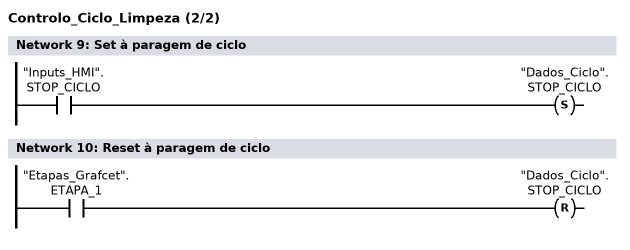
   RUNG wire#powerrail
      Contact( "Inputs_HMI".STOP_CICLO )
      S_Coil( "Dados_Ciclo".STOP_CICLO )
   END_RUNG
   // the same network as SCL:
   IF "Inputs_HMI".STOP_CICLO THEN "Dados_Ciclo".STOP_CICLO := TRUE; END_IF;
END_REGION

REGION Network 10: Reset à paragem de ciclo
   RUNG wire#powerrail
      Contact( "Etapas_Grafcet".ETAPA_1 )
      R_Coil( "Dados_Ciclo".STOP_CICLO )
   END_RUNG
   // the same network as SCL:
   IF "Etapas_Grafcet".ETAPA_1 THEN "Dados_Ciclo".STOP_CICLO := FALSE; END_IF;
END_REGION
END_FUNCTION

FUNCTION "Controlo_Pressostatos" : Void   // FC8, LAD
TITLE = Ao fim de 30s indica que atingiu setpoint de pressão
{ S7_Optimized_Access := 'TRUE' }
VERSION : 0.1
// stored: AutoNumber true, IsIECCheckEnabled false, SetENOAutomatically false, UDAEnableTagReadback false
BEGIN

REGION Network 1: Pressostato Filtro 1
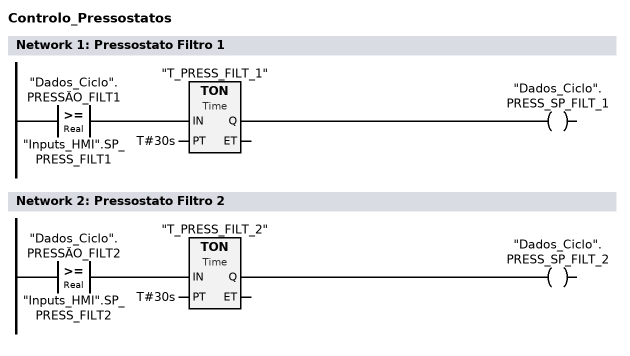
   RUNG wire#powerrail
      { S7_Templates := "SrcType := Real" } GE_Contact(in1 := "Dados_Ciclo".PRESSÃO_FILT1, in2 := "Inputs_HMI".SP_PRESS_FILT1)
      { S7_Templates := "time_type := Time" } "T_PRESS_FILT_1".TON(pt := T#30s, et =>)
      Coil( "Dados_Ciclo".PRESS_SP_FILT_1 )
   END_RUNG
   // the same network as SCL:
   "T_PRESS_FILT_1".TON(IN := "Dados_Ciclo".PRESSÃO_FILT1 >= "Inputs_HMI".SP_PRESS_FILT1, PT := T#30s);
   "Dados_Ciclo".PRESS_SP_FILT_1 := "T_PRESS_FILT_1".Q;
END_REGION

REGION Network 2: Pressostato Filtro 2
   RUNG wire#powerrail
      { S7_Templates := "SrcType := Real" } GE_Contact(in1 := "Dados_Ciclo".PRESSÃO_FILT2, in2 := "Inputs_HMI".SP_PRESS_FILT2)
      { S7_Templates := "time_type := Time" } "T_PRESS_FILT_2".TON(pt := T#30s, et =>)
      Coil( "Dados_Ciclo".PRESS_SP_FILT_2 )
   END_RUNG
   // the same network as SCL:
   "T_PRESS_FILT_2".TON(IN := "Dados_Ciclo".PRESSÃO_FILT2 >= "Inputs_HMI".SP_PRESS_FILT2, PT := T#30s);
   "Dados_Ciclo".PRESS_SP_FILT_2 := "T_PRESS_FILT_2".Q;
END_REGION
END_FUNCTION

FUNCTION "Saídas_Bombas" : Void   // FC3, LAD
{ S7_Optimized_Access := 'TRUE' }
VERSION : 0.1
// stored: AutoNumber true, IsIECCheckEnabled false, SetENOAutomatically false, UDAEnableTagReadback false
   VAR_TEMP
      BOMBA_1_VAR : Bool;
      BOMBA_2_VAR : Bool;
      BOMBA_3_RESERVA : Bool;
   END_VAR
BEGIN

REGION Network 1: Bomba 1 (com variador)
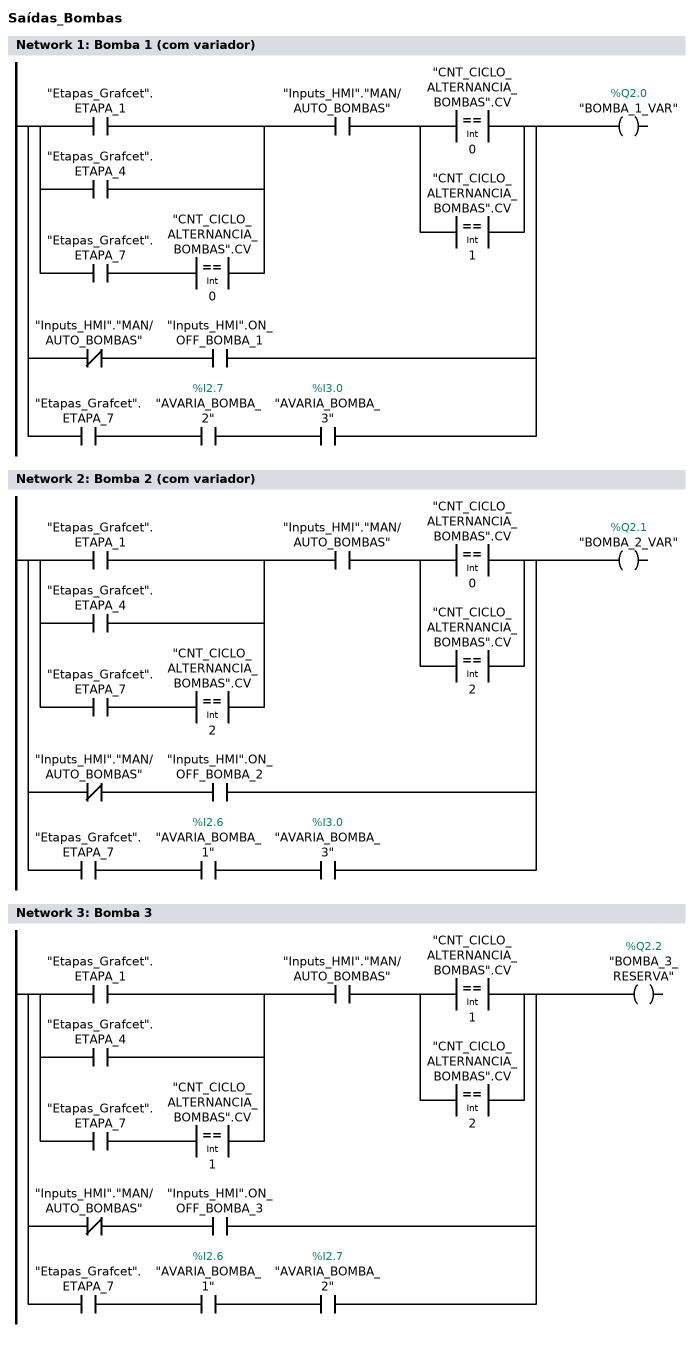
   RUNG wire#powerrail
      Contact( "Etapas_Grafcet".ETAPA_1 )
      wire#w1
      Contact( "Inputs_HMI"."MAN/AUTO_BOMBAS" )
      wire#w2
      { S7_Templates := "SrcType := Int" } EQ_Contact(in1 := "CNT_CICLO_ALTERNANCIA_BOMBAS".CV, in2 := 0)
      wire#w3
      Coil( "BOMBA_1_VAR" )
   END_RUNG
   RUNG wire#powerrail
      Contact( "Etapas_Grafcet".ETAPA_4 )
   END_RUNG wire#w1
   RUNG wire#powerrail
      Contact( "Etapas_Grafcet".ETAPA_7 )
      { S7_Templates := "SrcType := Int" } EQ_Contact(in1 := "CNT_CICLO_ALTERNANCIA_BOMBAS".CV, in2 := 0)
   END_RUNG wire#w1
   RUNG wire#w2
      { S7_Templates := "SrcType := Int" } EQ_Contact(in1 := "CNT_CICLO_ALTERNANCIA_BOMBAS".CV, in2 := 1)
   END_RUNG wire#w3
   RUNG wire#powerrail
      I_Contact( "Inputs_HMI"."MAN/AUTO_BOMBAS" )
      Contact( "Inputs_HMI".ON_OFF_BOMBA_1 )
   END_RUNG wire#w3
   RUNG wire#powerrail
      Contact( "Etapas_Grafcet".ETAPA_7 )
      Contact( "AVARIA_BOMBA_2" )
      Contact( "AVARIA_BOMBA_3" )
   END_RUNG wire#w3
   // the same network as SCL:
   "BOMBA_1_VAR" := (("Etapas_Grafcet".ETAPA_1 OR "Etapas_Grafcet".ETAPA_4 OR ("Etapas_Grafcet".ETAPA_7 AND ("CNT_CICLO_ALTERNANCIA_BOMBAS".CV = 0))) AND "Inputs_HMI"."MAN/AUTO_BOMBAS" AND (("CNT_CICLO_ALTERNANCIA_BOMBAS".CV = 0) OR ("CNT_CICLO_ALTERNANCIA_BOMBAS".CV = 1))) OR (NOT "Inputs_HMI"."MAN/AUTO_BOMBAS" AND "Inputs_HMI".ON_OFF_BOMBA_1) OR ("Etapas_Grafcet".ETAPA_7 AND "AVARIA_BOMBA_2" AND "AVARIA_BOMBA_3");
END_REGION

REGION Network 2: Bomba 2 (com variador)
   RUNG wire#powerrail
      Contact( "Etapas_Grafcet".ETAPA_1 )
      wire#w1
      Contact( "Inputs_HMI"."MAN/AUTO_BOMBAS" )
      wire#w2
      { S7_Templates := "SrcType := Int" } EQ_Contact(in1 := "CNT_CICLO_ALTERNANCIA_BOMBAS".CV, in2 := 0)
      wire#w3
      Coil( "BOMBA_2_VAR" )
   END_RUNG
   RUNG wire#powerrail
      Contact( "Etapas_Grafcet".ETAPA_4 )
   END_RUNG wire#w1
   RUNG wire#powerrail
      Contact( "Etapas_Grafcet".ETAPA_7 )
      { S7_Templates := "SrcType := Int" } EQ_Contact(in1 := "CNT_CICLO_ALTERNANCIA_BOMBAS".CV, in2 := 2)
   END_RUNG wire#w1
   RUNG wire#w2
      { S7_Templates := "SrcType := Int" } EQ_Contact(in1 := "CNT_CICLO_ALTERNANCIA_BOMBAS".CV, in2 := 2)
   END_RUNG wire#w3
   RUNG wire#powerrail
      I_Contact( "Inputs_HMI"."MAN/AUTO_BOMBAS" )
      Contact( "Inputs_HMI".ON_OFF_BOMBA_2 )
   END_RUNG wire#w3
   RUNG wire#powerrail
      Contact( "Etapas_Grafcet".ETAPA_7 )
      Contact( "AVARIA_BOMBA_1" )
      Contact( "AVARIA_BOMBA_3" )
   END_RUNG wire#w3
   // the same network as SCL:
   "BOMBA_2_VAR" := (("Etapas_Grafcet".ETAPA_1 OR "Etapas_Grafcet".ETAPA_4 OR ("Etapas_Grafcet".ETAPA_7 AND ("CNT_CICLO_ALTERNANCIA_BOMBAS".CV = 2))) AND "Inputs_HMI"."MAN/AUTO_BOMBAS" AND (("CNT_CICLO_ALTERNANCIA_BOMBAS".CV = 0) OR ("CNT_CICLO_ALTERNANCIA_BOMBAS".CV = 2))) OR (NOT "Inputs_HMI"."MAN/AUTO_BOMBAS" AND "Inputs_HMI".ON_OFF_BOMBA_2) OR ("Etapas_Grafcet".ETAPA_7 AND "AVARIA_BOMBA_1" AND "AVARIA_BOMBA_3");
END_REGION

REGION Network 3: Bomba 3
   RUNG wire#powerrail
      Contact( "Etapas_Grafcet".ETAPA_1 )
      wire#w1
      Contact( "Inputs_HMI"."MAN/AUTO_BOMBAS" )
      wire#w2
      { S7_Templates := "SrcType := Int" } EQ_Contact(in1 := "CNT_CICLO_ALTERNANCIA_BOMBAS".CV, in2 := 1)
      wire#w3
      Coil( "BOMBA_3_RESERVA" )
   END_RUNG
   RUNG wire#powerrail
      Contact( "Etapas_Grafcet".ETAPA_4 )
   END_RUNG wire#w1
   RUNG wire#powerrail
      Contact( "Etapas_Grafcet".ETAPA_7 )
      { S7_Templates := "SrcType := Int" } EQ_Contact(in1 := "CNT_CICLO_ALTERNANCIA_BOMBAS".CV, in2 := 1)
   END_RUNG wire#w1
   RUNG wire#w2
      { S7_Templates := "SrcType := Int" } EQ_Contact(in1 := "CNT_CICLO_ALTERNANCIA_BOMBAS".CV, in2 := 2)
   END_RUNG wire#w3
   RUNG wire#powerrail
      I_Contact( "Inputs_HMI"."MAN/AUTO_BOMBAS" )
      Contact( "Inputs_HMI".ON_OFF_BOMBA_3 )
   END_RUNG wire#w3
   RUNG wire#powerrail
      Contact( "Etapas_Grafcet".ETAPA_7 )
      Contact( "AVARIA_BOMBA_1" )
      Contact( "AVARIA_BOMBA_2" )
   END_RUNG wire#w3
   // the same network as SCL:
   "BOMBA_3_RESERVA" := (("Etapas_Grafcet".ETAPA_1 OR "Etapas_Grafcet".ETAPA_4 OR ("Etapas_Grafcet".ETAPA_7 AND ("CNT_CICLO_ALTERNANCIA_BOMBAS".CV = 1))) AND "Inputs_HMI"."MAN/AUTO_BOMBAS" AND (("CNT_CICLO_ALTERNANCIA_BOMBAS".CV = 1) OR ("CNT_CICLO_ALTERNANCIA_BOMBAS".CV = 2))) OR (NOT "Inputs_HMI"."MAN/AUTO_BOMBAS" AND "Inputs_HMI".ON_OFF_BOMBA_3) OR ("Etapas_Grafcet".ETAPA_7 AND "AVARIA_BOMBA_1" AND "AVARIA_BOMBA_2");
END_REGION
END_FUNCTION

FUNCTION "Saídas_EV_Filt1" : Void   // FC4, LAD
{ S7_Optimized_Access := 'TRUE' }
VERSION : 0.1
// stored: AutoNumber true, IsIECCheckEnabled false, SetENOAutomatically false, UDAEnableTagReadback false
BEGIN

REGION Network 1
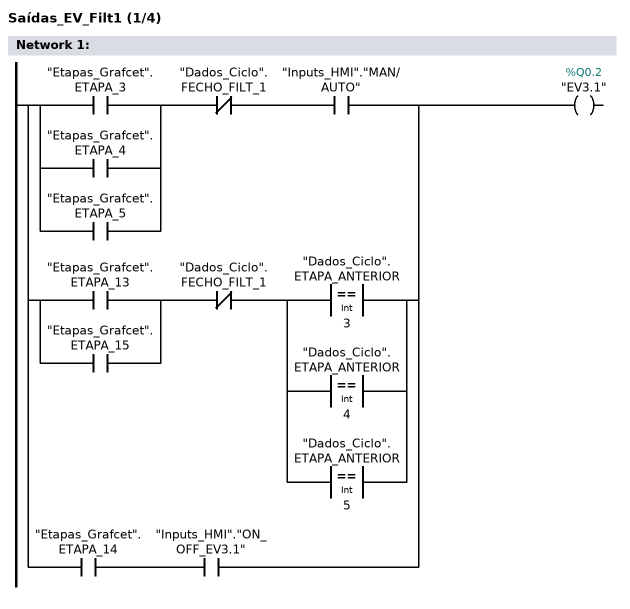
   RUNG wire#powerrail
      Contact( "Etapas_Grafcet".ETAPA_3 )
      wire#w1
      I_Contact( "Dados_Ciclo".FECHO_FILT_1 )
      Contact( "Inputs_HMI"."MAN/AUTO" )
      wire#w2
      Coil( "EV3.1" )
   END_RUNG
   RUNG wire#powerrail
      Contact( "Etapas_Grafcet".ETAPA_4 )
   END_RUNG wire#w1
   RUNG wire#powerrail
      Contact( "Etapas_Grafcet".ETAPA_5 )
   END_RUNG wire#w1
   RUNG wire#powerrail
      Contact( "Etapas_Grafcet".ETAPA_13 )
      wire#w3
      I_Contact( "Dados_Ciclo".FECHO_FILT_1 )
      wire#w4
      { S7_Templates := "SrcType := Int" } EQ_Contact(in1 := "Dados_Ciclo".ETAPA_ANTERIOR, in2 := 3)
   END_RUNG wire#w2
   RUNG wire#powerrail
      Contact( "Etapas_Grafcet".ETAPA_15 )
   END_RUNG wire#w3
   RUNG wire#w4
      { S7_Templates := "SrcType := Int" } EQ_Contact(in1 := "Dados_Ciclo".ETAPA_ANTERIOR, in2 := 4)
   END_RUNG wire#w2
   RUNG wire#w4
      { S7_Templates := "SrcType := Int" } EQ_Contact(in1 := "Dados_Ciclo".ETAPA_ANTERIOR, in2 := 5)
   END_RUNG wire#w2
   RUNG wire#powerrail
      Contact( "Etapas_Grafcet".ETAPA_14 )
      Contact( "Inputs_HMI"."ON_OFF_EV3.1" )
   END_RUNG wire#w2
   // the same network as SCL:
   "EV3.1" := (("Etapas_Grafcet".ETAPA_3 OR "Etapas_Grafcet".ETAPA_4 OR "Etapas_Grafcet".ETAPA_5) AND NOT "Dados_Ciclo".FECHO_FILT_1 AND "Inputs_HMI"."MAN/AUTO") OR (("Etapas_Grafcet".ETAPA_13 OR "Etapas_Grafcet".ETAPA_15) AND NOT "Dados_Ciclo".FECHO_FILT_1 AND (("Dados_Ciclo".ETAPA_ANTERIOR = 3) OR ("Dados_Ciclo".ETAPA_ANTERIOR = 4) OR ("Dados_Ciclo".ETAPA_ANTERIOR = 5))) OR ("Etapas_Grafcet".ETAPA_14 AND "Inputs_HMI"."ON_OFF_EV3.1");
END_REGION

REGION Network 2
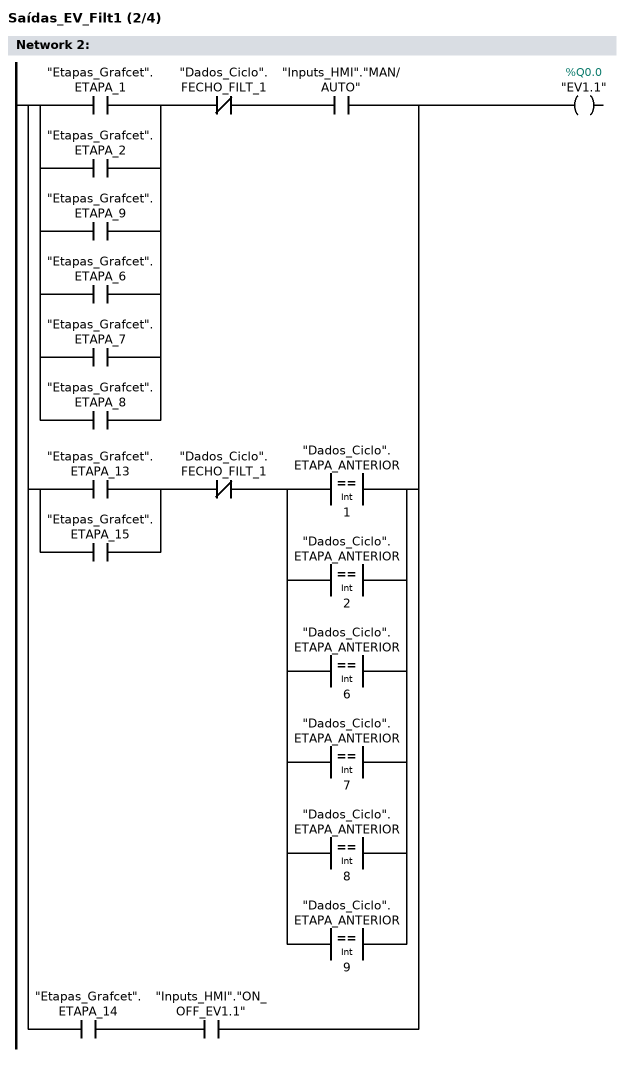
   RUNG wire#powerrail
      Contact( "Etapas_Grafcet".ETAPA_1 )
      wire#w1
      I_Contact( "Dados_Ciclo".FECHO_FILT_1 )
      Contact( "Inputs_HMI"."MAN/AUTO" )
      wire#w2
      Coil( "EV1.1" )
   END_RUNG
   RUNG wire#powerrail
      Contact( "Etapas_Grafcet".ETAPA_2 )
   END_RUNG wire#w1
   RUNG wire#powerrail
      Contact( "Etapas_Grafcet".ETAPA_9 )
   END_RUNG wire#w1
   RUNG wire#powerrail
      Contact( "Etapas_Grafcet".ETAPA_6 )
   END_RUNG wire#w1
   RUNG wire#powerrail
      Contact( "Etapas_Grafcet".ETAPA_7 )
   END_RUNG wire#w1
   RUNG wire#powerrail
      Contact( "Etapas_Grafcet".ETAPA_8 )
   END_RUNG wire#w1
   RUNG wire#powerrail
      Contact( "Etapas_Grafcet".ETAPA_13 )
      wire#w3
      I_Contact( "Dados_Ciclo".FECHO_FILT_1 )
      wire#w4
      { S7_Templates := "SrcType := Int" } EQ_Contact(in1 := "Dados_Ciclo".ETAPA_ANTERIOR, in2 := 1)
   END_RUNG wire#w2
   RUNG wire#powerrail
      Contact( "Etapas_Grafcet".ETAPA_15 )
   END_RUNG wire#w3
   RUNG wire#w4
      { S7_Templates := "SrcType := Int" } EQ_Contact(in1 := "Dados_Ciclo".ETAPA_ANTERIOR, in2 := 2)
   END_RUNG wire#w2
   RUNG wire#w4
      { S7_Templates := "SrcType := Int" } EQ_Contact(in1 := "Dados_Ciclo".ETAPA_ANTERIOR, in2 := 6)
   END_RUNG wire#w2
   RUNG wire#w4
      { S7_Templates := "SrcType := Int" } EQ_Contact(in1 := "Dados_Ciclo".ETAPA_ANTERIOR, in2 := 7)
   END_RUNG wire#w2
   RUNG wire#w4
      { S7_Templates := "SrcType := Int" } EQ_Contact(in1 := "Dados_Ciclo".ETAPA_ANTERIOR, in2 := 8)
   END_RUNG wire#w2
   RUNG wire#w4
      { S7_Templates := "SrcType := Int" } EQ_Contact(in1 := "Dados_Ciclo".ETAPA_ANTERIOR, in2 := 9)
   END_RUNG wire#w2
   RUNG wire#powerrail
      Contact( "Etapas_Grafcet".ETAPA_14 )
      Contact( "Inputs_HMI"."ON_OFF_EV1.1" )
   END_RUNG wire#w2
   // the same network as SCL:
   "EV1.1" := (("Etapas_Grafcet".ETAPA_1 OR "Etapas_Grafcet".ETAPA_2 OR "Etapas_Grafcet".ETAPA_9 OR "Etapas_Grafcet".ETAPA_6 OR "Etapas_Grafcet".ETAPA_7 OR "Etapas_Grafcet".ETAPA_8) AND NOT "Dados_Ciclo".FECHO_FILT_1 AND "Inputs_HMI"."MAN/AUTO") OR (("Etapas_Grafcet".ETAPA_13 OR "Etapas_Grafcet".ETAPA_15) AND NOT "Dados_Ciclo".FECHO_FILT_1 AND (("Dados_Ciclo".ETAPA_ANTERIOR = 1) OR ("Dados_Ciclo".ETAPA_ANTERIOR = 2) OR ("Dados_Ciclo".ETAPA_ANTERIOR = 6) OR ("Dados_Ciclo".ETAPA_ANTERIOR = 7) OR ("Dados_Ciclo".ETAPA_ANTERIOR = 8) OR ("Dados_Ciclo".ETAPA_ANTERIOR = 9))) OR ("Etapas_Grafcet".ETAPA_14 AND "Inputs_HMI"."ON_OFF_EV1.1");
END_REGION

REGION Network 3
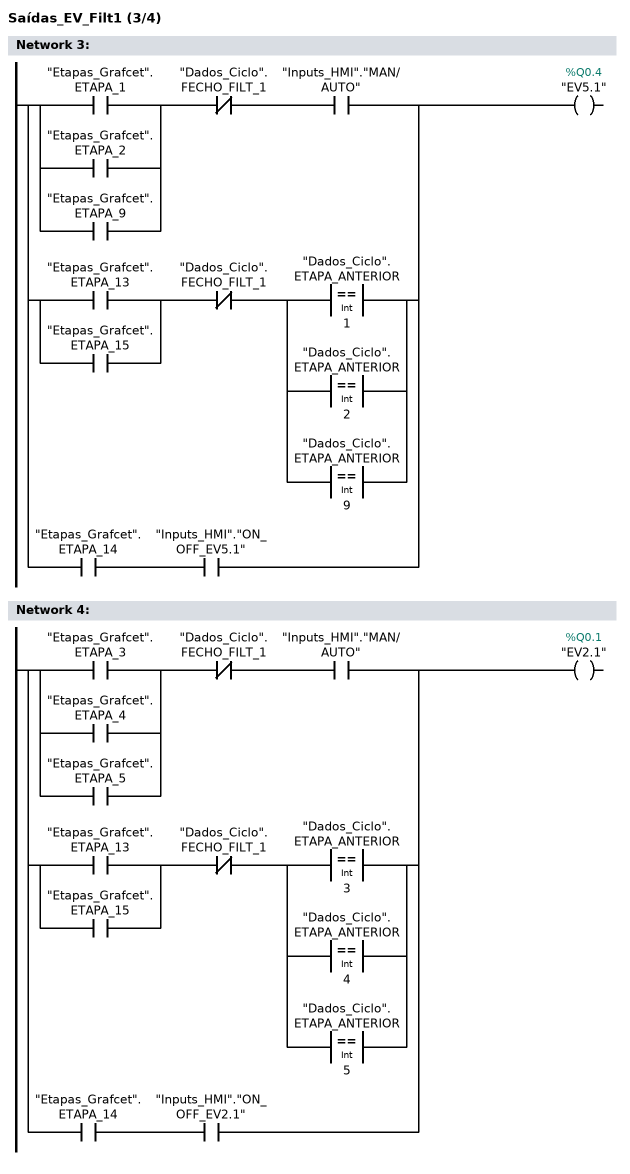
   RUNG wire#powerrail
      Contact( "Etapas_Grafcet".ETAPA_1 )
      wire#w1
      I_Contact( "Dados_Ciclo".FECHO_FILT_1 )
      Contact( "Inputs_HMI"."MAN/AUTO" )
      wire#w2
      Coil( "EV5.1" )
   END_RUNG
   RUNG wire#powerrail
      Contact( "Etapas_Grafcet".ETAPA_2 )
   END_RUNG wire#w1
   RUNG wire#powerrail
      Contact( "Etapas_Grafcet".ETAPA_9 )
   END_RUNG wire#w1
   RUNG wire#powerrail
      Contact( "Etapas_Grafcet".ETAPA_13 )
      wire#w3
      I_Contact( "Dados_Ciclo".FECHO_FILT_1 )
      wire#w4
      { S7_Templates := "SrcType := Int" } EQ_Contact(in1 := "Dados_Ciclo".ETAPA_ANTERIOR, in2 := 1)
   END_RUNG wire#w2
   RUNG wire#powerrail
      Contact( "Etapas_Grafcet".ETAPA_15 )
   END_RUNG wire#w3
   RUNG wire#w4
      { S7_Templates := "SrcType := Int" } EQ_Contact(in1 := "Dados_Ciclo".ETAPA_ANTERIOR, in2 := 2)
   END_RUNG wire#w2
   RUNG wire#w4
      { S7_Templates := "SrcType := Int" } EQ_Contact(in1 := "Dados_Ciclo".ETAPA_ANTERIOR, in2 := 9)
   END_RUNG wire#w2
   RUNG wire#powerrail
      Contact( "Etapas_Grafcet".ETAPA_14 )
      Contact( "Inputs_HMI"."ON_OFF_EV5.1" )
   END_RUNG wire#w2
   // the same network as SCL:
   "EV5.1" := (("Etapas_Grafcet".ETAPA_1 OR "Etapas_Grafcet".ETAPA_2 OR "Etapas_Grafcet".ETAPA_9) AND NOT "Dados_Ciclo".FECHO_FILT_1 AND "Inputs_HMI"."MAN/AUTO") OR (("Etapas_Grafcet".ETAPA_13 OR "Etapas_Grafcet".ETAPA_15) AND NOT "Dados_Ciclo".FECHO_FILT_1 AND (("Dados_Ciclo".ETAPA_ANTERIOR = 1) OR ("Dados_Ciclo".ETAPA_ANTERIOR = 2) OR ("Dados_Ciclo".ETAPA_ANTERIOR = 9))) OR ("Etapas_Grafcet".ETAPA_14 AND "Inputs_HMI"."ON_OFF_EV5.1");
END_REGION

REGION Network 4
   RUNG wire#powerrail
      Contact( "Etapas_Grafcet".ETAPA_3 )
      wire#w1
      I_Contact( "Dados_Ciclo".FECHO_FILT_1 )
      Contact( "Inputs_HMI"."MAN/AUTO" )
      wire#w2
      Coil( "EV2.1" )
   END_RUNG
   RUNG wire#powerrail
      Contact( "Etapas_Grafcet".ETAPA_4 )
   END_RUNG wire#w1
   RUNG wire#powerrail
      Contact( "Etapas_Grafcet".ETAPA_5 )
   END_RUNG wire#w1
   RUNG wire#powerrail
      Contact( "Etapas_Grafcet".ETAPA_13 )
      wire#w3
      I_Contact( "Dados_Ciclo".FECHO_FILT_1 )
      wire#w4
      { S7_Templates := "SrcType := Int" } EQ_Contact(in1 := "Dados_Ciclo".ETAPA_ANTERIOR, in2 := 3)
   END_RUNG wire#w2
   RUNG wire#powerrail
      Contact( "Etapas_Grafcet".ETAPA_15 )
   END_RUNG wire#w3
   RUNG wire#w4
      { S7_Templates := "SrcType := Int" } EQ_Contact(in1 := "Dados_Ciclo".ETAPA_ANTERIOR, in2 := 4)
   END_RUNG wire#w2
   RUNG wire#w4
      { S7_Templates := "SrcType := Int" } EQ_Contact(in1 := "Dados_Ciclo".ETAPA_ANTERIOR, in2 := 5)
   END_RUNG wire#w2
   RUNG wire#powerrail
      Contact( "Etapas_Grafcet".ETAPA_14 )
      Contact( "Inputs_HMI"."ON_OFF_EV2.1" )
   END_RUNG wire#w2
   // the same network as SCL:
   "EV2.1" := (("Etapas_Grafcet".ETAPA_3 OR "Etapas_Grafcet".ETAPA_4 OR "Etapas_Grafcet".ETAPA_5) AND NOT "Dados_Ciclo".FECHO_FILT_1 AND "Inputs_HMI"."MAN/AUTO") OR (("Etapas_Grafcet".ETAPA_13 OR "Etapas_Grafcet".ETAPA_15) AND NOT "Dados_Ciclo".FECHO_FILT_1 AND (("Dados_Ciclo".ETAPA_ANTERIOR = 3) OR ("Dados_Ciclo".ETAPA_ANTERIOR = 4) OR ("Dados_Ciclo".ETAPA_ANTERIOR = 5))) OR ("Etapas_Grafcet".ETAPA_14 AND "Inputs_HMI"."ON_OFF_EV2.1");
END_REGION

REGION Network 5
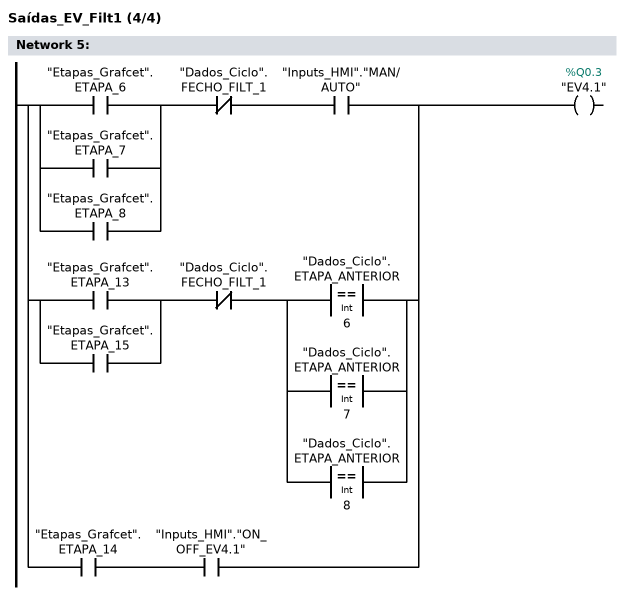
   RUNG wire#powerrail
      Contact( "Etapas_Grafcet".ETAPA_6 )
      wire#w1
      I_Contact( "Dados_Ciclo".FECHO_FILT_1 )
      Contact( "Inputs_HMI"."MAN/AUTO" )
      wire#w2
      Coil( "EV4.1" )
   END_RUNG
   RUNG wire#powerrail
      Contact( "Etapas_Grafcet".ETAPA_7 )
   END_RUNG wire#w1
   RUNG wire#powerrail
      Contact( "Etapas_Grafcet".ETAPA_8 )
   END_RUNG wire#w1
   RUNG wire#powerrail
      Contact( "Etapas_Grafcet".ETAPA_13 )
      wire#w3
      I_Contact( "Dados_Ciclo".FECHO_FILT_1 )
      wire#w4
      { S7_Templates := "SrcType := Int" } EQ_Contact(in1 := "Dados_Ciclo".ETAPA_ANTERIOR, in2 := 6)
   END_RUNG wire#w2
   RUNG wire#powerrail
      Contact( "Etapas_Grafcet".ETAPA_15 )
   END_RUNG wire#w3
   RUNG wire#w4
      { S7_Templates := "SrcType := Int" } EQ_Contact(in1 := "Dados_Ciclo".ETAPA_ANTERIOR, in2 := 7)
   END_RUNG wire#w2
   RUNG wire#w4
      { S7_Templates := "SrcType := Int" } EQ_Contact(in1 := "Dados_Ciclo".ETAPA_ANTERIOR, in2 := 8)
   END_RUNG wire#w2
   RUNG wire#powerrail
      Contact( "Etapas_Grafcet".ETAPA_14 )
      Contact( "Inputs_HMI"."ON_OFF_EV4.1" )
   END_RUNG wire#w2
   // the same network as SCL:
   "EV4.1" := (("Etapas_Grafcet".ETAPA_6 OR "Etapas_Grafcet".ETAPA_7 OR "Etapas_Grafcet".ETAPA_8) AND NOT "Dados_Ciclo".FECHO_FILT_1 AND "Inputs_HMI"."MAN/AUTO") OR (("Etapas_Grafcet".ETAPA_13 OR "Etapas_Grafcet".ETAPA_15) AND NOT "Dados_Ciclo".FECHO_FILT_1 AND (("Dados_Ciclo".ETAPA_ANTERIOR = 6) OR ("Dados_Ciclo".ETAPA_ANTERIOR = 7) OR ("Dados_Ciclo".ETAPA_ANTERIOR = 8))) OR ("Etapas_Grafcet".ETAPA_14 AND "Inputs_HMI"."ON_OFF_EV4.1");
END_REGION
END_FUNCTION

FUNCTION "Saídas_EV_Filt2" : Void   // FC5, LAD
{ S7_Optimized_Access := 'TRUE' }
VERSION : 0.1
// stored: AutoNumber true, IsIECCheckEnabled false, SetENOAutomatically false, UDAEnableTagReadback false
BEGIN

REGION Network 1
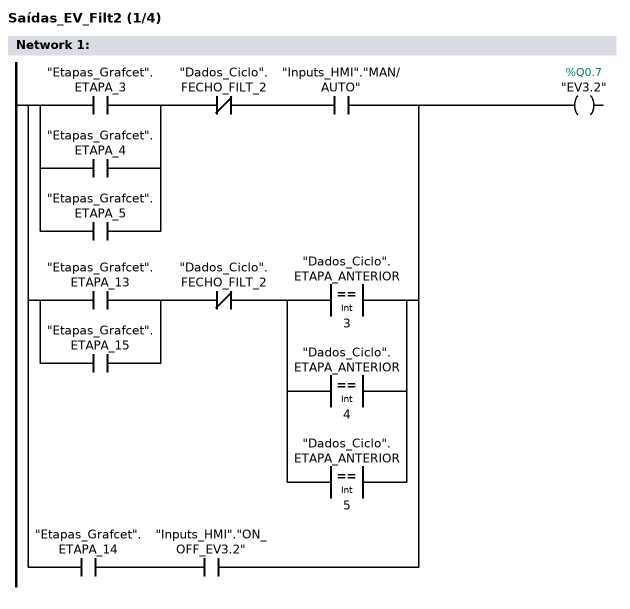
   RUNG wire#powerrail
      Contact( "Etapas_Grafcet".ETAPA_3 )
      wire#w1
      I_Contact( "Dados_Ciclo".FECHO_FILT_2 )
      Contact( "Inputs_HMI"."MAN/AUTO" )
      wire#w2
      Coil( "EV3.2" )
   END_RUNG
   RUNG wire#powerrail
      Contact( "Etapas_Grafcet".ETAPA_4 )
   END_RUNG wire#w1
   RUNG wire#powerrail
      Contact( "Etapas_Grafcet".ETAPA_5 )
   END_RUNG wire#w1
   RUNG wire#powerrail
      Contact( "Etapas_Grafcet".ETAPA_13 )
      wire#w3
      I_Contact( "Dados_Ciclo".FECHO_FILT_2 )
      wire#w4
      { S7_Templates := "SrcType := Int" } EQ_Contact(in1 := "Dados_Ciclo".ETAPA_ANTERIOR, in2 := 3)
   END_RUNG wire#w2
   RUNG wire#powerrail
      Contact( "Etapas_Grafcet".ETAPA_15 )
   END_RUNG wire#w3
   RUNG wire#w4
      { S7_Templates := "SrcType := Int" } EQ_Contact(in1 := "Dados_Ciclo".ETAPA_ANTERIOR, in2 := 4)
   END_RUNG wire#w2
   RUNG wire#w4
      { S7_Templates := "SrcType := Int" } EQ_Contact(in1 := "Dados_Ciclo".ETAPA_ANTERIOR, in2 := 5)
   END_RUNG wire#w2
   RUNG wire#powerrail
      Contact( "Etapas_Grafcet".ETAPA_14 )
      Contact( "Inputs_HMI"."ON_OFF_EV3.2" )
   END_RUNG wire#w2
   // the same network as SCL:
   "EV3.2" := (("Etapas_Grafcet".ETAPA_3 OR "Etapas_Grafcet".ETAPA_4 OR "Etapas_Grafcet".ETAPA_5) AND NOT "Dados_Ciclo".FECHO_FILT_2 AND "Inputs_HMI"."MAN/AUTO") OR (("Etapas_Grafcet".ETAPA_13 OR "Etapas_Grafcet".ETAPA_15) AND NOT "Dados_Ciclo".FECHO_FILT_2 AND (("Dados_Ciclo".ETAPA_ANTERIOR = 3) OR ("Dados_Ciclo".ETAPA_ANTERIOR = 4) OR ("Dados_Ciclo".ETAPA_ANTERIOR = 5))) OR ("Etapas_Grafcet".ETAPA_14 AND "Inputs_HMI"."ON_OFF_EV3.2");
END_REGION

REGION Network 2
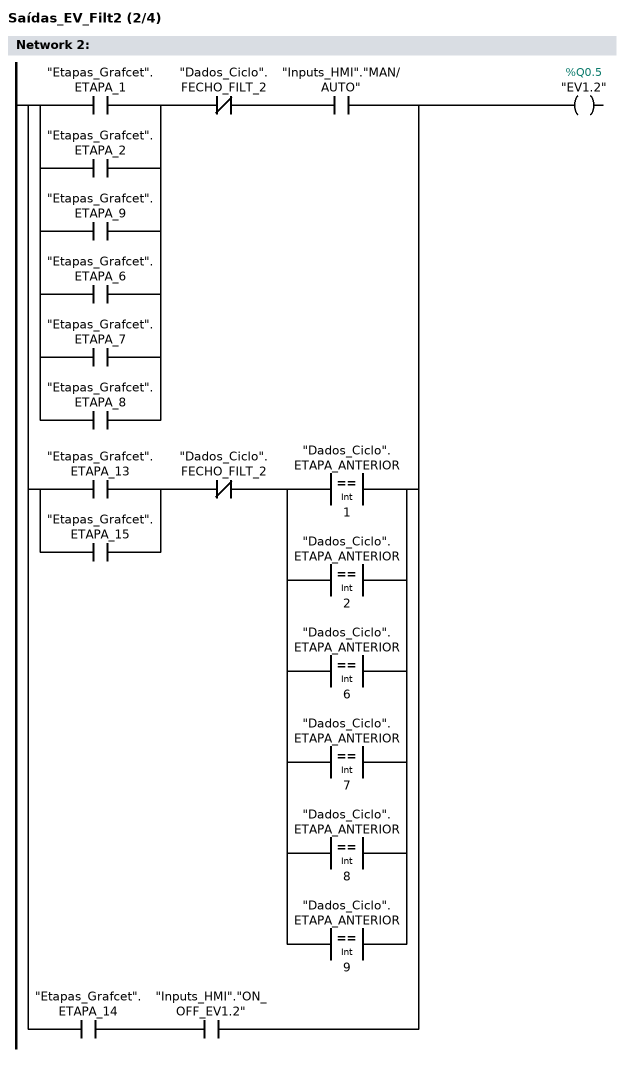
   RUNG wire#powerrail
      Contact( "Etapas_Grafcet".ETAPA_1 )
      wire#w1
      I_Contact( "Dados_Ciclo".FECHO_FILT_2 )
      Contact( "Inputs_HMI"."MAN/AUTO" )
      wire#w2
      Coil( "EV1.2" )
   END_RUNG
   RUNG wire#powerrail
      Contact( "Etapas_Grafcet".ETAPA_2 )
   END_RUNG wire#w1
   RUNG wire#powerrail
      Contact( "Etapas_Grafcet".ETAPA_9 )
   END_RUNG wire#w1
   RUNG wire#powerrail
      Contact( "Etapas_Grafcet".ETAPA_6 )
   END_RUNG wire#w1
   RUNG wire#powerrail
      Contact( "Etapas_Grafcet".ETAPA_7 )
   END_RUNG wire#w1
   RUNG wire#powerrail
      Contact( "Etapas_Grafcet".ETAPA_8 )
   END_RUNG wire#w1
   RUNG wire#powerrail
      Contact( "Etapas_Grafcet".ETAPA_13 )
      wire#w3
      I_Contact( "Dados_Ciclo".FECHO_FILT_2 )
      wire#w4
      { S7_Templates := "SrcType := Int" } EQ_Contact(in1 := "Dados_Ciclo".ETAPA_ANTERIOR, in2 := 1)
   END_RUNG wire#w2
   RUNG wire#powerrail
      Contact( "Etapas_Grafcet".ETAPA_15 )
   END_RUNG wire#w3
   RUNG wire#w4
      { S7_Templates := "SrcType := Int" } EQ_Contact(in1 := "Dados_Ciclo".ETAPA_ANTERIOR, in2 := 2)
   END_RUNG wire#w2
   RUNG wire#w4
      { S7_Templates := "SrcType := Int" } EQ_Contact(in1 := "Dados_Ciclo".ETAPA_ANTERIOR, in2 := 6)
   END_RUNG wire#w2
   RUNG wire#w4
      { S7_Templates := "SrcType := Int" } EQ_Contact(in1 := "Dados_Ciclo".ETAPA_ANTERIOR, in2 := 7)
   END_RUNG wire#w2
   RUNG wire#w4
      { S7_Templates := "SrcType := Int" } EQ_Contact(in1 := "Dados_Ciclo".ETAPA_ANTERIOR, in2 := 8)
   END_RUNG wire#w2
   RUNG wire#w4
      { S7_Templates := "SrcType := Int" } EQ_Contact(in1 := "Dados_Ciclo".ETAPA_ANTERIOR, in2 := 9)
   END_RUNG wire#w2
   RUNG wire#powerrail
      Contact( "Etapas_Grafcet".ETAPA_14 )
      Contact( "Inputs_HMI"."ON_OFF_EV1.2" )
   END_RUNG wire#w2
   // the same network as SCL:
   "EV1.2" := (("Etapas_Grafcet".ETAPA_1 OR "Etapas_Grafcet".ETAPA_2 OR "Etapas_Grafcet".ETAPA_9 OR "Etapas_Grafcet".ETAPA_6 OR "Etapas_Grafcet".ETAPA_7 OR "Etapas_Grafcet".ETAPA_8) AND NOT "Dados_Ciclo".FECHO_FILT_2 AND "Inputs_HMI"."MAN/AUTO") OR (("Etapas_Grafcet".ETAPA_13 OR "Etapas_Grafcet".ETAPA_15) AND NOT "Dados_Ciclo".FECHO_FILT_2 AND (("Dados_Ciclo".ETAPA_ANTERIOR = 1) OR ("Dados_Ciclo".ETAPA_ANTERIOR = 2) OR ("Dados_Ciclo".ETAPA_ANTERIOR = 6) OR ("Dados_Ciclo".ETAPA_ANTERIOR = 7) OR ("Dados_Ciclo".ETAPA_ANTERIOR = 8) OR ("Dados_Ciclo".ETAPA_ANTERIOR = 9))) OR ("Etapas_Grafcet".ETAPA_14 AND "Inputs_HMI"."ON_OFF_EV1.2");
END_REGION

REGION Network 3
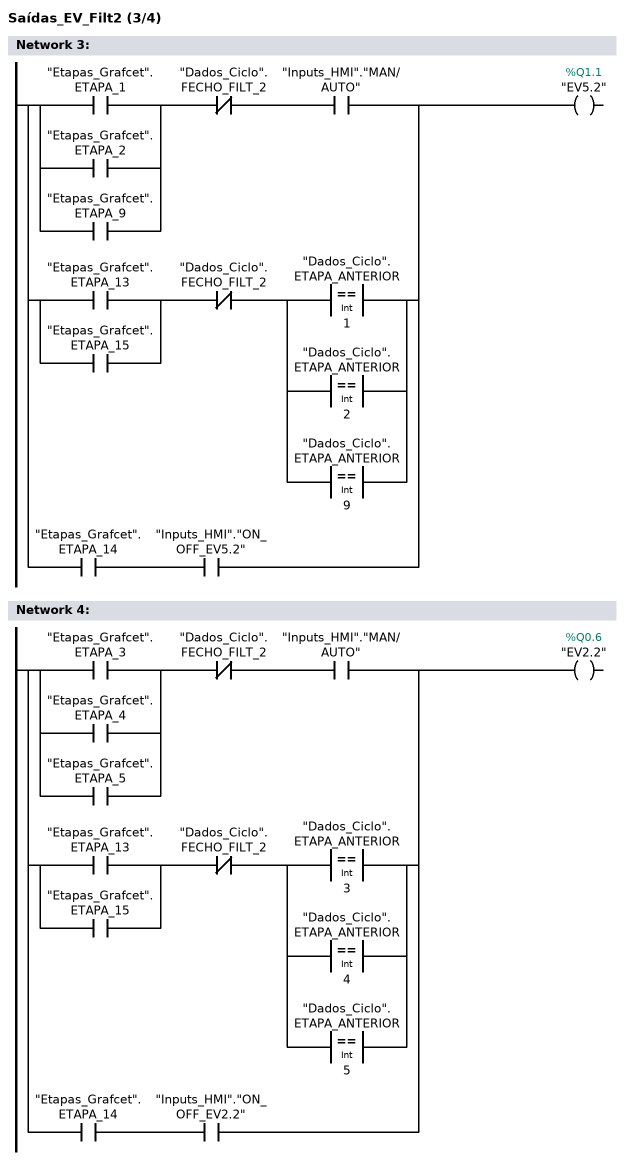
   RUNG wire#powerrail
      Contact( "Etapas_Grafcet".ETAPA_1 )
      wire#w1
      I_Contact( "Dados_Ciclo".FECHO_FILT_2 )
      Contact( "Inputs_HMI"."MAN/AUTO" )
      wire#w2
      Coil( "EV5.2" )
   END_RUNG
   RUNG wire#powerrail
      Contact( "Etapas_Grafcet".ETAPA_2 )
   END_RUNG wire#w1
   RUNG wire#powerrail
      Contact( "Etapas_Grafcet".ETAPA_9 )
   END_RUNG wire#w1
   RUNG wire#powerrail
      Contact( "Etapas_Grafcet".ETAPA_13 )
      wire#w3
      I_Contact( "Dados_Ciclo".FECHO_FILT_2 )
      wire#w4
      { S7_Templates := "SrcType := Int" } EQ_Contact(in1 := "Dados_Ciclo".ETAPA_ANTERIOR, in2 := 1)
   END_RUNG wire#w2
   RUNG wire#powerrail
      Contact( "Etapas_Grafcet".ETAPA_15 )
   END_RUNG wire#w3
   RUNG wire#w4
      { S7_Templates := "SrcType := Int" } EQ_Contact(in1 := "Dados_Ciclo".ETAPA_ANTERIOR, in2 := 2)
   END_RUNG wire#w2
   RUNG wire#w4
      { S7_Templates := "SrcType := Int" } EQ_Contact(in1 := "Dados_Ciclo".ETAPA_ANTERIOR, in2 := 9)
   END_RUNG wire#w2
   RUNG wire#powerrail
      Contact( "Etapas_Grafcet".ETAPA_14 )
      Contact( "Inputs_HMI"."ON_OFF_EV5.2" )
   END_RUNG wire#w2
   // the same network as SCL:
   "EV5.2" := (("Etapas_Grafcet".ETAPA_1 OR "Etapas_Grafcet".ETAPA_2 OR "Etapas_Grafcet".ETAPA_9) AND NOT "Dados_Ciclo".FECHO_FILT_2 AND "Inputs_HMI"."MAN/AUTO") OR (("Etapas_Grafcet".ETAPA_13 OR "Etapas_Grafcet".ETAPA_15) AND NOT "Dados_Ciclo".FECHO_FILT_2 AND (("Dados_Ciclo".ETAPA_ANTERIOR = 1) OR ("Dados_Ciclo".ETAPA_ANTERIOR = 2) OR ("Dados_Ciclo".ETAPA_ANTERIOR = 9))) OR ("Etapas_Grafcet".ETAPA_14 AND "Inputs_HMI"."ON_OFF_EV5.2");
END_REGION

REGION Network 4
   RUNG wire#powerrail
      Contact( "Etapas_Grafcet".ETAPA_3 )
      wire#w1
      I_Contact( "Dados_Ciclo".FECHO_FILT_2 )
      Contact( "Inputs_HMI"."MAN/AUTO" )
      wire#w2
      Coil( "EV2.2" )
   END_RUNG
   RUNG wire#powerrail
      Contact( "Etapas_Grafcet".ETAPA_4 )
   END_RUNG wire#w1
   RUNG wire#powerrail
      Contact( "Etapas_Grafcet".ETAPA_5 )
   END_RUNG wire#w1
   RUNG wire#powerrail
      Contact( "Etapas_Grafcet".ETAPA_13 )
      wire#w3
      I_Contact( "Dados_Ciclo".FECHO_FILT_2 )
      wire#w4
      { S7_Templates := "SrcType := Int" } EQ_Contact(in1 := "Dados_Ciclo".ETAPA_ANTERIOR, in2 := 3)
   END_RUNG wire#w2
   RUNG wire#powerrail
      Contact( "Etapas_Grafcet".ETAPA_15 )
   END_RUNG wire#w3
   RUNG wire#w4
      { S7_Templates := "SrcType := Int" } EQ_Contact(in1 := "Dados_Ciclo".ETAPA_ANTERIOR, in2 := 4)
   END_RUNG wire#w2
   RUNG wire#w4
      { S7_Templates := "SrcType := Int" } EQ_Contact(in1 := "Dados_Ciclo".ETAPA_ANTERIOR, in2 := 5)
   END_RUNG wire#w2
   RUNG wire#powerrail
      Contact( "Etapas_Grafcet".ETAPA_14 )
      Contact( "Inputs_HMI"."ON_OFF_EV2.2" )
   END_RUNG wire#w2
   // the same network as SCL:
   "EV2.2" := (("Etapas_Grafcet".ETAPA_3 OR "Etapas_Grafcet".ETAPA_4 OR "Etapas_Grafcet".ETAPA_5) AND NOT "Dados_Ciclo".FECHO_FILT_2 AND "Inputs_HMI"."MAN/AUTO") OR (("Etapas_Grafcet".ETAPA_13 OR "Etapas_Grafcet".ETAPA_15) AND NOT "Dados_Ciclo".FECHO_FILT_2 AND (("Dados_Ciclo".ETAPA_ANTERIOR = 3) OR ("Dados_Ciclo".ETAPA_ANTERIOR = 4) OR ("Dados_Ciclo".ETAPA_ANTERIOR = 5))) OR ("Etapas_Grafcet".ETAPA_14 AND "Inputs_HMI"."ON_OFF_EV2.2");
END_REGION

REGION Network 5
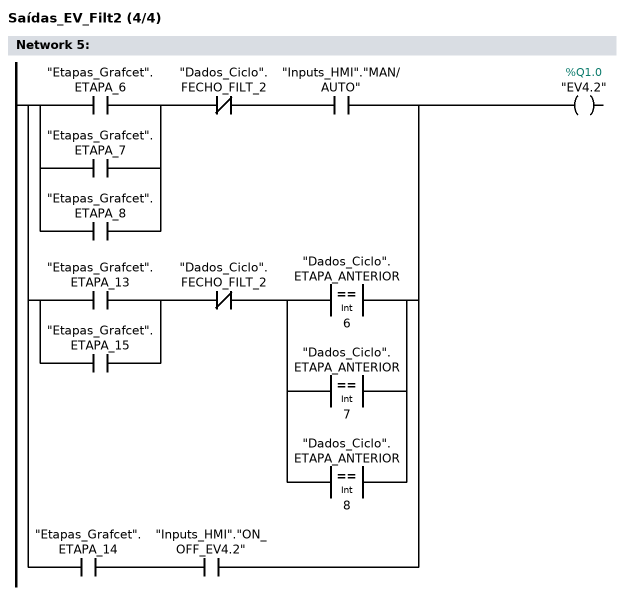
   RUNG wire#powerrail
      Contact( "Etapas_Grafcet".ETAPA_6 )
      wire#w1
      I_Contact( "Dados_Ciclo".FECHO_FILT_2 )
      Contact( "Inputs_HMI"."MAN/AUTO" )
      wire#w2
      Coil( "EV4.2" )
   END_RUNG
   RUNG wire#powerrail
      Contact( "Etapas_Grafcet".ETAPA_7 )
   END_RUNG wire#w1
   RUNG wire#powerrail
      Contact( "Etapas_Grafcet".ETAPA_8 )
   END_RUNG wire#w1
   RUNG wire#powerrail
      Contact( "Etapas_Grafcet".ETAPA_13 )
      wire#w3
      I_Contact( "Dados_Ciclo".FECHO_FILT_2 )
      wire#w4
      { S7_Templates := "SrcType := Int" } EQ_Contact(in1 := "Dados_Ciclo".ETAPA_ANTERIOR, in2 := 6)
   END_RUNG wire#w2
   RUNG wire#powerrail
      Contact( "Etapas_Grafcet".ETAPA_15 )
   END_RUNG wire#w3
   RUNG wire#w4
      { S7_Templates := "SrcType := Int" } EQ_Contact(in1 := "Dados_Ciclo".ETAPA_ANTERIOR, in2 := 7)
   END_RUNG wire#w2
   RUNG wire#w4
      { S7_Templates := "SrcType := Int" } EQ_Contact(in1 := "Dados_Ciclo".ETAPA_ANTERIOR, in2 := 8)
   END_RUNG wire#w2
   RUNG wire#powerrail
      Contact( "Etapas_Grafcet".ETAPA_14 )
      Contact( "Inputs_HMI"."ON_OFF_EV4.2" )
   END_RUNG wire#w2
   // the same network as SCL:
   "EV4.2" := (("Etapas_Grafcet".ETAPA_6 OR "Etapas_Grafcet".ETAPA_7 OR "Etapas_Grafcet".ETAPA_8) AND NOT "Dados_Ciclo".FECHO_FILT_2 AND "Inputs_HMI"."MAN/AUTO") OR (("Etapas_Grafcet".ETAPA_13 OR "Etapas_Grafcet".ETAPA_15) AND NOT "Dados_Ciclo".FECHO_FILT_2 AND (("Dados_Ciclo".ETAPA_ANTERIOR = 6) OR ("Dados_Ciclo".ETAPA_ANTERIOR = 7) OR ("Dados_Ciclo".ETAPA_ANTERIOR = 8))) OR ("Etapas_Grafcet".ETAPA_14 AND "Inputs_HMI"."ON_OFF_EV4.2");
END_REGION
END_FUNCTION

FUNCTION "UV" : Void   // FC15, LAD
{ S7_Optimized_Access := 'TRUE' }
VERSION : 0.1
// stored: AutoNumber true, IsIECCheckEnabled false, SetENOAutomatically false, UDAEnableTagReadback false
   VAR_TEMP
      sr_ultravioleta : Bool;
   END_VAR
BEGIN

REGION Network 1
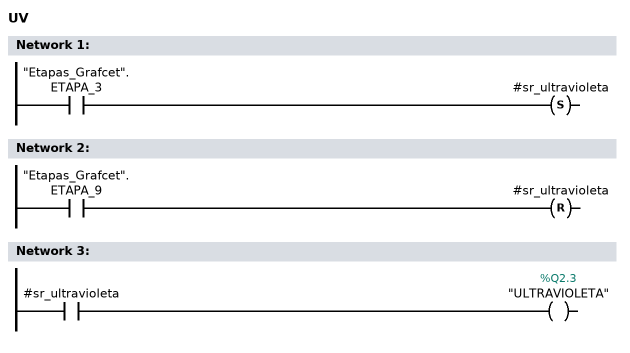
   RUNG wire#powerrail
      Contact( "Etapas_Grafcet".ETAPA_3 )
      S_Coil( #sr_ultravioleta )
   END_RUNG
   // the same network as SCL:
   IF "Etapas_Grafcet".ETAPA_3 THEN #sr_ultravioleta := TRUE; END_IF;
END_REGION

REGION Network 2
   RUNG wire#powerrail
      Contact( "Etapas_Grafcet".ETAPA_9 )
      R_Coil( #sr_ultravioleta )
   END_RUNG
   // the same network as SCL:
   IF "Etapas_Grafcet".ETAPA_9 THEN #sr_ultravioleta := FALSE; END_IF;
END_REGION

REGION Network 3
   RUNG wire#powerrail
      Contact( #sr_ultravioleta )
      Coil( "ULTRAVIOLETA" )
   END_RUNG
   // the same network as SCL:
   "ULTRAVIOLETA" := #sr_ultravioleta;
END_REGION
END_FUNCTION

FUNCTION "FC33_Auxiliary_Memories" : Void
{ S7_Optimized_Access := 'TRUE' }
VERSION : 0.0
   VAR_TEMP 
      p_carr : DInt;
      TempDInt : DInt;
      TempDInt2 : DInt;
      TempDInt_MLC : DInt;
   END_VAR


BEGIN
	//Auxiliary memories pt.2
	//***********************
	(*
	//
	//CONDIZIONI PER EMERGENZA MACCHINA
	"EmergencyCondition" := (NOT "Main_EMG") OR
	                        (NOT "Thermic") OR  //EmergencyCode = 62
	                        "Alarm2" OR
	                        "Bumper";
	//
	*)
	//GESTIONE MALFUNZIONAMENTI INVERTER
	//FAULT (anomalia)
	IF ("Inverter_Data".U201.actual_fault = 16#0000) AND
	    ("Inverter_Data".U221.actual_fault = 16#0000) AND
	    ("Inverter_Data".U241.actual_fault = 16#0000) AND
	    ("Inverter_Data".U261.actual_fault = 16#0000) AND
	    ("Inverter_Data".U321.actual_fault = 16#0000) THEN
	    //    
	    "InverterFault" := 0;
	    "InverterFail" := 0;
	ELSE
	    "InverterFault" := 1;
	END_IF;
	//ALARM (avviso)
	IF ("Inverter_Data".U201.actual_alarm = 16#0000) AND
	    ("Inverter_Data".U221.actual_alarm = 16#0000) AND
	    ("Inverter_Data".U241.actual_alarm = 16#0000) AND
	    ("Inverter_Data".U261.actual_alarm = 16#0000) AND
	    ("Inverter_Data".U321.actual_alarm = 16#0000) THEN
	    //    
	    "InverterAlarm" := 0;
	ELSE    //copio il codice avviso (per poi visualizzarlo su HMI se persiste)
	    "Inverter_Alarms".U201_alarm := "Inverter_Data".U201.actual_alarm;
	    "Inverter_Alarms".U221_alarm := "Inverter_Data".U221.actual_alarm;
	    "Inverter_Alarms".U241_alarm := "Inverter_Data".U241.actual_alarm;
	    "Inverter_Alarms".U261_alarm := "Inverter_Data".U261.actual_alarm;
	    "Inverter_Alarms".U321_alarm := "Inverter_Data".U321.actual_alarm;
	    //    
	    "InverterAlarm" := 1;
	END_IF;
	//
	IF "Reset" THEN
	    "Inverter_Alarms".U201_alarm := 0;
	    "Inverter_Alarms".U221_alarm := 0;
	    "Inverter_Alarms".U241_alarm := 0;
	    "Inverter_Alarms".U261_alarm := 0;
	    "Inverter_Alarms".U321_alarm := 0;
	END_IF;
	//
	//Nel caso di "avvisi" attivo l'allarme solo se persistono per 5 secondi
	//
	IF ("InverterFault" OR "Timer".T200.Q) THEN
	    "InverterFail" := 1;
	    "DB23_AlarmProgram".dbx0_4 := 1;
	END_IF;
	//RESET (ACK)
	IF "Timer".T4.Q THEN
	    "U201_Ack" := 1;
	    "U221_Ack" := 1;
	    "U241_Ack" := 1;
	    "U261_Ack" := 1;
	    "U321_Ack" := 1;
	ELSE
	    "U201_Ack" := 0;
	    "U221_Ack" := 0;
	    "U241_Ack" := 0;
	    "U261_Ack" := 0;
	    "U321_Ack" := 0;
	END_IF;
	//
	//GESTIONE CELLA DI CARICO
	//************************
	(**)
	"CELLA" := "MB_REG1".A08R.REG_0; //(FC320_PID)
	//"CELLA" := 450; //(FC320_PID)
	//Reset cella
	IF "ResetLoadCell" THEN
	    "DB215_ProgramData".Offset_cella := "CELLA" + "DB215_ProgramData".ValOffsetCella;
	END_IF;
	//
	//APPOGGIO PER GRAFICO PID
	//*****
	//ROSA
	"DB100_Display".CELLA := ("CELLA" - 100) / 8;  //cella carico
	//ROSSO
	"DB100_Display".SETPOINT := ("DB320_PID".PID.setPointShow - 100) / 8;  //sp calcolato (cella)
	//VERDE
	"DB100_Display".PROP := (1 * DINT_TO_INT("DB320_PID".PID.proporzionale)) / 2;  //proporzionale
	//GIALLO
	"DB100_Display"."INT" := (1 * DINT_TO_INT("DB320_PID".PID.integrativo)) / 3;  //integrale
	//
	//AZZURRO
	"DB100_Display".FREQ_TIRO := (REAL_TO_INT("Inverter_Data".U241.setpoint)) / 30;  //integrale
	//AZZURRO
	"DB100_Display".FREQ_PRES := (REAL_TO_INT("Inverter_Data".U261.setpoint)) / 30;  //integrale
	//
	(*
	//
	//MOTORIZZAZIONI
	//Passi carrello + rotazione
	IF "DB230_Parameters".MotorType THEN
	    //SEW
	    "DB20_DisplaySysdata".dbd0 := 3730; 
	    "DB20_DisplaySysdata".dbd80 := 3180;
	ELSE //STD
	    "DB20_DisplaySysdata".dbd0 := 3330;
	    "DB20_DisplaySysdata".dbd80 := 7230; //enc.non integrato (P1)
	END_IF;
	//
	//Costanti per proporzioni velocità 
	"DB215_ProgramData".PropArmMax := 1770; //braccio@15rpm
	"DB215_ProgramData".PropCarrMax := 1933; //carrello@7.2m/min=120mm/s
	//
	//GESTIONE BRACCIO
	//****************
	//Zona sicurezza braccio (fuori ingombro)
	//
	IF "DB09_ArmPos".dbw34 > 3200 OR "DB09_ArmPos".dbw34 < 460 THEN
	    "SafetyPhase" := 1;
	ELSE
	    "SafetyPhase" := 0;
	END_IF;
	//
	//FASE DI TAGLIO
	//IF "DB09_ArmPos".dbw34 > 350 AND "DB09_ArmPos".dbw34 < 380 THEN
	IF ("DB09_ArmPos".dbw34 > ("DB230_Parameters".Cut_Phase - "DB20_DisplaySysdata".dbw84)) AND
	   ("DB09_ArmPos".dbw34 < ("DB230_Parameters".Cut_Phase + "DB20_DisplaySysdata".dbw84)) THEN
	    "CutPhase" := 1;
	ELSE
	    "CutPhase" := 0;
	END_IF;
	//
	//Velocità rotazione
	"DB215_ProgramData".RotSpeed := USINT_TO_INT("DB216_ActiveRecipe".Recipe.RotSpeed) * "DB215_ProgramData".PropArmMax / 15;
	//
	//Calcoli per decelerazione
	//Durata di un giro in ms in base alla velocità (60.000 msec / velocità in rpm)
	(*
	IF NOT "DB215_ProgramData".ActiveRecipeMLC THEN
	    "DB215_ProgramData".RoundTime := 60000 / USINT_TO_UINT("DB216_ActiveRecipe".Recipe.RotSpeed);
	ELSE
	    "DB215_ProgramData".RoundTime := 60000 / USINT_TO_UINT("DB216_ActiveRecipe".Recipe.MLC_L9.RotSpeed);
	END_IF;
	*)
	"DIAGNOSTICA".int_19 := INT_TO_UINT("DIAGNOSTICA".int_09);
	"DB215_ProgramData".RoundTime := 6000 / "DIAGNOSTICA".int_19; //decimi
	//Aumento il tempo in cui iniziare la decelerazione al diminuire della velocità (ci mette meno a fermarsi)
	//
	(*
	IF NOT "DB215_ProgramData".ActiveRecipeMLC THEN
	    #TempDInt := 125 - 5 * "DB216_ActiveRecipe".Recipe.RotSpeed; //(% di tempo giro) [(50:90) per (15:7)rpm]
	ELSE
	    #TempDInt := 125 - 5 * "DB216_ActiveRecipe".Recipe.MLC_L9.RotSpeed; //(% di tempo giro) [(50:90) per (15:7)rpm]
	END_IF;
	*)
	#TempDInt := 1250 - 5 * ("DIAGNOSTICA".int_19); //(% di tempo giro) [(50:90) per (15:7)rpm]
	#TempDInt2 := 60000 / "DIAGNOSTICA".int_19;//"DB215_ProgramData".RoundTime;    //T_giro
	"DB215_ProgramData".LastRoundTime := DINT_TO_UINT((#TempDInt * #TempDInt2) / 100);  //millisec
	//
	//GESTIONE CARRELLO
	//*****************
	//Direzione conteggio
	IF "FlagCarUp" THEN
	    "DB215_ProgramData".EncCarrDir := 1; //direzione conteggio UP
	ELSE
	    "DB215_ProgramData".EncCarrDir := -1; //direzione conteggio DOWN
	END_IF;
	//
	//Velocità salita/discesa
	#TempDInt := USINT_TO_DINT("DB216_ActiveRecipe".Recipe.CarSpeedUp) * "DB215_ProgramData".PropCarrMax / 72;
	"DB215_ProgramData".CarSpeedUp := DINT_TO_INT(#TempDInt);
	//
	#TempDInt := USINT_TO_DINT("DB216_ActiveRecipe".Recipe.CarSpeedDw) * "DB215_ProgramData".PropCarrMax / 72;
	"DB215_ProgramData".CarSpeedDw := DINT_TO_INT(#TempDInt);
	//
	//POSIZIONAMENTI CARRELLO
	//Passo [mm/1000p]
	#p_carr := "DB20_DisplaySysdata".dbd0;
	//
	//Altimetro
	#TempDInt := UINT_TO_DINT("DB216_ActiveRecipe".Recipe.Altimeter - 50) * 10000;
	"DB215_ProgramData".Altimeter_Pulses := DINT_TO_INT(#TempDInt / #p_carr);
	//
	//Ritardo fotocellula [ciclo STD; per MLC vedi FC33]
	//(se ho attivo il pressore considero lo spessore di circa 8 cm in meno del piatto)
	IF "DB216_ActiveRecipe".Recipe.PresserEnable THEN
	    IF "DB216_ActiveRecipe".Recipe.PhotDelay >= 8 THEN
	        #TempDInt := USINT_TO_DINT("DB216_ActiveRecipe".Recipe.PhotDelay - 8) * 10000;
	    ELSE
	        #TempDInt := USINT_TO_DINT("DB216_ActiveRecipe".Recipe.PhotDelay) * 10000;
	    END_IF;
	ELSE
	    #TempDInt := USINT_TO_DINT("DB216_ActiveRecipe".Recipe.PhotDelay) * 10000;
	END_IF;
	"DB215_ProgramData".PhotDelay_Pulses := DINT_TO_INT(#TempDInt / #p_carr);
	//
	//Giri rinforzo
	#TempDInt := USINT_TO_DINT("DB216_ActiveRecipe".Recipe.ReinforceHeight) * 10000;
	"DB215_ProgramData".Reinforce_Pulses := DINT_TO_INT(#TempDInt / #p_carr);
	//Discesa carrello per top
	#TempDInt := INT_TO_DINT("DB230_Parameters".TopCarrDescent) * 10000;
	"DB215_ProgramData".TopFall_Pulses := DINT_TO_INT(#TempDInt / #p_carr);
	//MLC
	//Forzamento a zero dell'ultimo strato (sempre in basso)
	"DB216_ActiveRecipe".Recipe.MLC_L9.Height := 0;
	//
	//Altezza strati (in base allo step del ciclo MLC) - Carica dati dello strato successivo
	IF "DB215_ProgramData".ActiveRecipeMLC THEN
	    CASE "DB200_Supervisor".State_Auto OF
	        15:
	            #TempDInt_MLC := UINT_TO_DINT("DB216_ActiveRecipe".Recipe.MLC_L1.Height) * 10000;
	            "DB215_ProgramData".MLC_HeightPulses := DINT_TO_INT(#TempDInt_MLC / #p_carr);
	//-----------------------------------------------------------------------------------------------            
	        212:
	            #TempDInt_MLC := UINT_TO_DINT("DB216_ActiveRecipe".Recipe.MLC_L2.Height) * 10000;
	            "DB215_ProgramData".MLC_HeightPulses := DINT_TO_INT(#TempDInt_MLC / #p_carr);
	//-----------------------------------------------------------------------------------------------            
	        220:
	            #TempDInt_MLC := UINT_TO_DINT("DB216_ActiveRecipe".Recipe.MLC_L2.Height) * 10000;
	            "DB215_ProgramData".MLC_HeightPulses := DINT_TO_INT(#TempDInt_MLC / #p_carr);
	        222:
	            #TempDInt_MLC := UINT_TO_DINT("DB216_ActiveRecipe".Recipe.MLC_L3.Height) * 10000;
	            "DB215_ProgramData".MLC_HeightPulses := DINT_TO_INT(#TempDInt_MLC / #p_carr);
	//-----------------------------------------------------------------------------------------------             
	        230:
	            #TempDInt_MLC := UINT_TO_DINT("DB216_ActiveRecipe".Recipe.MLC_L3.Height) * 10000;
	            "DB215_ProgramData".MLC_HeightPulses := DINT_TO_INT(#TempDInt_MLC / #p_carr);
	        232:
	            #TempDInt_MLC := UINT_TO_DINT("DB216_ActiveRecipe".Recipe.MLC_L4.Height) * 10000;
	            "DB215_ProgramData".MLC_HeightPulses := DINT_TO_INT(#TempDInt_MLC / #p_carr);
	//----------------------------------------------------------------------------------------------- 
	        240:
	            #TempDInt_MLC := UINT_TO_DINT("DB216_ActiveRecipe".Recipe.MLC_L4.Height) * 10000;
	            "DB215_ProgramData".MLC_HeightPulses := DINT_TO_INT(#TempDInt_MLC / #p_carr);
	        242:
	            #TempDInt_MLC := UINT_TO_DINT("DB216_ActiveRecipe".Recipe.MLC_L5.Height - 50) * 10000;
	            "DB215_ProgramData".MLC_HeightPulses := DINT_TO_INT(#TempDInt_MLC / #p_carr);
	//-----------------------------------------------------------------------------------------------     
	        255:
	            #TempDInt_MLC := UINT_TO_DINT("DB216_ActiveRecipe".Recipe.MLC_L6.Height) * 10000;
	            "DB215_ProgramData".MLC_HeightPulses := DINT_TO_INT(#TempDInt_MLC / #p_carr);
	//-----------------------------------------------------------------------------------------------    
	        260:
	            #TempDInt_MLC := UINT_TO_DINT("DB216_ActiveRecipe".Recipe.MLC_L6.Height) * 10000;
	            "DB215_ProgramData".MLC_HeightPulses := DINT_TO_INT(#TempDInt_MLC / #p_carr);
	        262:
	            #TempDInt_MLC := UINT_TO_DINT("DB216_ActiveRecipe".Recipe.MLC_L7.Height) * 10000;
	            "DB215_ProgramData".MLC_HeightPulses := DINT_TO_INT(#TempDInt_MLC / #p_carr);
	//-----------------------------------------------------------------------------------------------
	        270:
	            #TempDInt_MLC := UINT_TO_DINT("DB216_ActiveRecipe".Recipe.MLC_L7.Height) * 10000;
	            "DB215_ProgramData".MLC_HeightPulses := DINT_TO_INT(#TempDInt_MLC / #p_carr);
	        272:
	            #TempDInt_MLC := UINT_TO_DINT("DB216_ActiveRecipe".Recipe.MLC_L8.Height) * 10000;
	            "DB215_ProgramData".MLC_HeightPulses := DINT_TO_INT(#TempDInt_MLC / #p_carr);
	//-----------------------------------------------------------------------------------------------
	        280:
	            #TempDInt_MLC := UINT_TO_DINT("DB216_ActiveRecipe".Recipe.MLC_L8.Height) * 10000;
	            "DB215_ProgramData".MLC_HeightPulses := DINT_TO_INT(#TempDInt_MLC / #p_carr);
	        282:
	            #TempDInt_MLC := UINT_TO_DINT("DB216_ActiveRecipe".Recipe.MLC_L9.Height) * 10000;
	            "DB215_ProgramData".MLC_HeightPulses := DINT_TO_INT(#TempDInt_MLC / #p_carr);
	    END_CASE;
	   //
	END_IF;
	//
	//Lettura posizione carrello
	"DIAGNOSTICA".dint_01 := ("Enc_Carr" * #p_carr) / 10000;
	//
	//GESTIONE CICLO AUTOMATICO
	//*************************
	"ActiveCycle" := ("DB200_Supervisor".State_Auto >= 10); // <> 0);
	//
	//RESET CICLO (PULSANTE HMI) - SOLO MACCHINA
	"DB100_Display".CycleResetEnable := ("DB200_Supervisor".State_Stop = 170 AND
	(NOT "CutPhase" OR NOT "CarriageDown" //OR
	//(LPAS_enable AND NOT "CutArmBack")
	OR "ActiveCycle"));
	//
	//RESET CICLO MACCHINA
	IF "Reset" AND "Stop_state" THEN
	    "DB200_Supervisor".State_Auto := 0;
	END_IF;
	//
	//TIPO CICLO (con/senza top per Rototech3000)
	//
	IF "DB216_ActiveRecipe".Recipe.Cycle >= 3 THEN
	    "DB216_ActiveRecipe".Recipe.Cycle := 0;
	END_IF;
	//Con MLC non ha senso parlare di ciclo economico (solo waterproof)
	IF "DB215_ProgramData".ActiveRecipeMLC THEN
	    IF "DB216_ActiveRecipe".Recipe.Cycle >= 2 THEN
	        "DB216_ActiveRecipe".Recipe.Cycle := 0;
	    END_IF;
	END_IF;
	//No top
	IF "DB216_ActiveRecipe".Recipe.Cycle = 0 THEN
	    "DB03_Machine".TopBefore := 0;
	    "DB03_Machine".TopWaterP := 0;
	END_IF;
	//Top waterproof
	IF "DB216_ActiveRecipe".Recipe.Cycle = 1 THEN
	    "DB03_Machine".TopBefore := 0;
	    "DB03_Machine".TopWaterP := 1;
	END_IF;
	//Top dustproof (top before)
	IF "DB216_ActiveRecipe".Recipe.Cycle = 2 THEN
	    "DB03_Machine".TopBefore := 1;
	    "DB03_Machine".TopWaterP := 0;
	END_IF;
	//
	//RICETTE
	//Confronto ricette su HMI (modificabile) e PLC (salvata)
	IF (%DB216.DBD0 <> %DB229.DBD0 OR
	    %DB216.DBD4 <> %DB229.DBD4 OR
	    %DB216.DBD8 <> %DB229.DBD8 OR
	    %DB216.DBD12 <> %DB229.DBD12 OR
	    %DB216.DBD16 <> %DB229.DBD16 OR
	    %DB216.DBD20 <> %DB229.DBD20 OR
	    %DB216.DBD24 <> %DB229.DBD24 OR
	    %DB216.DBD28 <> %DB229.DBD28 OR
	    %DB216.DBD32 <> %DB229.DBD32 OR
	    %DB216.DBD36 <> %DB229.DBD36 OR
	    %DB216.DBD40 <> %DB229.DBD40 OR
	    %DB216.DBD44 <> %DB229.DBD44 OR
	    %DB216.DBD48 <> %DB229.DBD48 OR
	    %DB216.DBD52 <> %DB229.DBD52 OR
	    %DB216.DBD56 <> %DB229.DBD56 OR
	    %DB216.DBD60 <> %DB229.DBD60 OR
	    %DB216.DBD64 <> %DB229.DBD64 OR
	    %DB216.DBD68 <> %DB229.DBD68 OR
	    %DB216.DBD72 <> %DB229.DBD72 OR
	    %DB216.DBD76 <> %DB229.DBD76 OR
	    %DB216.DBD80 <> %DB229.DBD80 OR
	    %DB216.DBD84 <> %DB229.DBD84 OR
	    %DB216.DBD88 <> %DB229.DBD88 OR
	    %DB216.DBD92 <> %DB229.DBD92 OR
	    %DB216.DBD96 <> %DB229.DBD96 OR
	    %DB216.DBD100 <> %DB229.DBD100 OR
	    %DB216.DBD104 <> %DB229.DBD104 OR
	    %DB216.DBD108 <> %DB229.DBD108 OR
	    %DB216.DBD112 <> %DB229.DBD112 OR
	    %DB216.DBD116 <> %DB229.DBD116 OR
	    %DB216.DBD120 <> %DB229.DBD120 OR
	    %DB216.DBD124 <> %DB229.DBD124 OR
	    %DB216.DBD128 <> %DB229.DBD128 OR
	    %DB216.DBD132 <> %DB229.DBD132 OR
	    %DB216.DBD136 <> %DB229.DBD136 OR
	    %DB216.DBD140 <> %DB229.DBD140 OR
	    %DB216.DBD144 <> %DB229.DBD144 OR
	    %DB216.DBD148 <> %DB229.DBD148 OR
	    %DB216.DBD152 <> %DB229.DBD152 OR
	    %DB216.DBD156 <> %DB229.DBD156)
	THEN
	    "DB215_ProgramData".RecipeModified := 1;
	ELSE
	    "DB215_ProgramData".RecipeModified := 0;
	END_IF;
	//******************************************
	//LIMITI
	//Tiro
	IF ("DB216_ActiveRecipe".Recipe.StretchDwRounds < 0) THEN
	    "DB216_ActiveRecipe".Recipe.StretchDwRounds := 0;
	ELSIF ("DB216_ActiveRecipe".Recipe.StretchDwRounds > 100) THEN
	    "DB216_ActiveRecipe".Recipe.StretchDwRounds := 100;
	END_IF;
	//Forzamento del valore di tiro giri bassi su altri valori
	IF NOT "DB100_Display".TiroMultipleVal THEN
	    IF "DB216_ActiveRecipe".Recipe.StretchDwRounds <> "DB216_ActiveRecipe".Recipe.StretchUpward THEN
	        "DB216_ActiveRecipe".Recipe.StretchUpward := "DB216_ActiveRecipe".Recipe.StretchDwRounds;
	    END_IF;
	    IF "DB216_ActiveRecipe".Recipe.StretchDwRounds <> "DB216_ActiveRecipe".Recipe.StretchUpRounds THEN
	        "DB216_ActiveRecipe".Recipe.StretchUpRounds := "DB216_ActiveRecipe".Recipe.StretchDwRounds;
	    END_IF;
	    IF "DB216_ActiveRecipe".Recipe.StretchDwRounds <> "DB216_ActiveRecipe".Recipe.StretchDownward THEN
	        "DB216_ActiveRecipe".Recipe.StretchDownward := "DB216_ActiveRecipe".Recipe.StretchDwRounds;
	    END_IF;
	END_IF;
	//Prestiro
	IF ("DB216_ActiveRecipe".Recipe.Prestretch < 150) THEN
	    "DB216_ActiveRecipe".Recipe.Prestretch := 150;
	ELSIF ("DB216_ActiveRecipe".Recipe.Prestretch > 400) THEN
	    "DB216_ActiveRecipe".Recipe.Prestretch := 400;
	END_IF;
	// Velocità braccio
	IF ("DB216_ActiveRecipe".Recipe.RotSpeed < 7) THEN
	    "DB216_ActiveRecipe".Recipe.RotSpeed := 7;
	ELSIF ("DB216_ActiveRecipe".Recipe.RotSpeed > 15) THEN
	    "DB216_ActiveRecipe".Recipe.RotSpeed := 15;
	END_IF;
	// Velocità carrello
	IF ("DB216_ActiveRecipe".Recipe.CarSpeedUp < 25) THEN
	    "DB216_ActiveRecipe".Recipe.CarSpeedUp := 25;
	ELSIF ("DB216_ActiveRecipe".Recipe.CarSpeedUp > 72) THEN
	    "DB216_ActiveRecipe".Recipe.CarSpeedUp := 72;
	END_IF;
	IF ("DB216_ActiveRecipe".Recipe.CarSpeedDw < 25) THEN
	    "DB216_ActiveRecipe".Recipe.CarSpeedDw := 25;
	ELSIF ("DB216_ActiveRecipe".Recipe.CarSpeedDw > 72) THEN
	    "DB216_ActiveRecipe".Recipe.CarSpeedDw := 72;
	END_IF;
	//******************************************
	*)
END_FUNCTION

FUNCTION "Alarmes_Disparos_2" : Void
{ S7_Optimized_Access := 'TRUE' }
VERSION : 0.1

BEGIN
	"Alarmes".ALARMES_1.%X3 := "BS001A_DISPARO";
	"Alarmes".ALARMES_1.%X4 := "BS001B_DISPARO";
	"Alarmes".ALARMES_1.%X5 := "MX201_DISPARO";
	"Alarmes".ALARMES_1.%X6 := "BH201_DISPARO";
	"Alarmes".ALARMES_1.%X7 := "MX301_DISPARO";
	"Alarmes".ALARMES_1.%X8 := "BM401_DISPARO";
	"Alarmes".ALARMES_1.%X9 := "BS501_DISPARO";
	"Alarmes".ALARMES_1.%X10 := "MX601_DISPARO";
	"Alarmes".ALARMES_1.%X11 := "BD601_DISPARO";
	"Alarmes".ALARMES_1.%X12 := "BD602_DISPARO";
	"Alarmes".ALARMES_1.%X13 := "MX603_DISPARO";
	"Alarmes".ALARMES_1.%X14 := "BD603_DISPARO";
	"Alarmes".ALARMES_1.%X15 := "MX604_DISPARO";
	"Alarmes".ALARMES_2.%X0 := "BD604_DISPARO";
	"Alarmes".ALARMES_2.%X1 := "MX605_DISPARO";
	"Alarmes".ALARMES_2.%X2 := "BD605_DISPARO";
	"Alarmes".ALARMES_2.%X3 := "DISPARO_DIF_3Q1_32";
	"Alarmes".ALARMES_2.%X4 := "DISPARO_DIFERENCIAL_3Q3";
	"Alarmes".ALARMES_2.%X5 := "DISPARO_DIFERENCIAL_4Q1_4Q2";
	"Alarmes".ALARMES_2.%X6 := NOT "FALHA_24VDC";
	"Alarmes".ALARMES_2.%X7 := "FALHA_220VAC";
	"Alarmes".ALARMES_2.%X8 := "FALHA_24VAC";
	
	
	
	
	
	
	
	
	
	
	
	
	
	
	
END_FUNCTION

FUNCTION "Alarmes" : Void
{ S7_Optimized_Access := 'TRUE' }
VERSION : 0.1

BEGIN
	//Alarmes filtro 1
	//
	REGION ALARME_V1.1
	    IF "T_ABERTURA_EV1.1_HMI".Q AND NOT "EV1.1_ABERTA" THEN  //Válvula não abriu
	        "Estados_HMI".ALARMES_LISTA_1.%X0 := TRUE;
	    ELSE
	        "Estados_HMI".ALARMES_LISTA_1.%X0 := FALSE;
	    END_IF;
	    
	    
	    IF "T_ABERTURA_EV1.1_HMI".Q AND "EV1.1_ABERTA" AND "EV1.1_FECHADA" THEN  //Avaria fim de curso de fecho
	        "Estados_HMI".ALARMES_LISTA_1.%X1 := TRUE;
	    ELSE
	        "Estados_HMI".ALARMES_LISTA_1.%X1 := FALSE;
	    END_IF;
	    
	    
	    IF "T_FECHO_EV1.1_HMI".Q AND NOT "EV1.1_FECHADA" THEN  //Válvula não fechou
	        "Estados_HMI".ALARMES_LISTA_1.%X2 := TRUE;
	    ELSE
	        "Estados_HMI".ALARMES_LISTA_1.%X2 := FALSE;
	    END_IF;
	    
	    
	    IF "T_FECHO_EV1.1_HMI".Q AND "EV1.1_ABERTA" AND "EV1.1_FECHADA" THEN  //Avaria fim de curso de abertura
	        "Estados_HMI".ALARMES_LISTA_1.%X3 := TRUE;
	    ELSE
	        "Estados_HMI".ALARMES_LISTA_1.%X3 := FALSE;
	    END_IF;
	END_REGION
	REGION ALARME_V2.1
	    IF "T_ABERTURA_EV2.1_HMI".Q AND NOT "EV2.1_ABERTA" THEN  //Válvula não abriu
	        "Estados_HMI".ALARMES_LISTA_1.%X4 := TRUE;
	    ELSE
	        "Estados_HMI".ALARMES_LISTA_1.%X4 := FALSE;
	    END_IF;
	    
	    
	    IF "T_ABERTURA_EV2.1_HMI".Q AND "EV2.1_ABERTA" AND "EV2.1_FECHADA" THEN  //Avaria fim de curso de fecho
	        "Estados_HMI".ALARMES_LISTA_1.%X5 := TRUE;
	    ELSE
	        "Estados_HMI".ALARMES_LISTA_1.%X5 := FALSE;
	    END_IF;
	    
	    
	    IF "T_FECHO_EV2.1_HMI".Q AND NOT "EV2.1_FECHADA" THEN  //Válvula não fechou
	        "Estados_HMI".ALARMES_LISTA_1.%X6 := TRUE;
	    ELSE
	        "Estados_HMI".ALARMES_LISTA_1.%X6 := FALSE;
	    END_IF;
	    
	    
	    IF "T_FECHO_EV2.1_HMI".Q AND "EV2.1_ABERTA" AND "EV2.1_FECHADA" THEN  //Avaria fim de curso de abertura
	        "Estados_HMI".ALARMES_LISTA_1.%X7 := TRUE;
	    ELSE
	        "Estados_HMI".ALARMES_LISTA_1.%X7 := FALSE;
	    END_IF;
	END_REGION
	REGION ALARME_V3.1
	    IF "T_ABERTURA_EV3.1_HMI".Q AND NOT "EV3.1_ABERTA" THEN  //Válvula não abriu
	        "Estados_HMI".ALARMES_LISTA_1.%X8 := TRUE;
	    ELSE
	        "Estados_HMI".ALARMES_LISTA_1.%X8 := FALSE;
	    END_IF;
	    
	    
	    IF "T_ABERTURA_EV3.1_HMI".Q AND "EV3.1_ABERTA" AND "EV3.1_FECHADA" THEN  //Avaria fim de curso de fecho
	        "Estados_HMI".ALARMES_LISTA_1.%X9 := TRUE;
	    ELSE
	        "Estados_HMI".ALARMES_LISTA_1.%X9 := FALSE;
	    END_IF;
	    
	    
	    IF "T_FECHO_EV3.1_HMI".Q AND NOT "EV3.1_FECHADA" THEN  //Válvula não fechou
	        "Estados_HMI".ALARMES_LISTA_1.%X10 := TRUE;
	    ELSE
	        "Estados_HMI".ALARMES_LISTA_1.%X10 := FALSE;
	    END_IF;
	    
	    
	    IF "T_FECHO_EV3.1_HMI".Q AND "EV3.1_ABERTA" AND "EV3.1_FECHADA" THEN  //Avaria fim de curso de abertura
	        "Estados_HMI".ALARMES_LISTA_1.%X11 := TRUE;
	    ELSE
	        "Estados_HMI".ALARMES_LISTA_1.%X11 := FALSE;
	    END_IF;
	END_REGION
	REGION ALARME_V4.1
	    IF "T_ABERTURA_EV4.1_HMI".Q AND NOT "EV4.1_ABERTA" THEN  //Válvula não abriu
	        "Estados_HMI".ALARMES_LISTA_1.%X12 := TRUE;
	    ELSE
	        "Estados_HMI".ALARMES_LISTA_1.%X12 := FALSE;
	    END_IF;
	    
	    
	    IF "T_ABERTURA_EV4.1_HMI".Q AND "EV4.1_ABERTA" AND "EV4.1_FECHADA" THEN  //Avaria fim de curso de fecho
	        "Estados_HMI".ALARMES_LISTA_1.%X13 := TRUE;
	    ELSE
	        "Estados_HMI".ALARMES_LISTA_1.%X13 := FALSE;
	    END_IF;
	    
	    
	    IF "T_FECHO_EV4.1_HMI".Q AND NOT "EV4.1_FECHADA" THEN  //Válvula não fechou
	        "Estados_HMI".ALARMES_LISTA_1.%X14 := TRUE;
	    ELSE
	        "Estados_HMI".ALARMES_LISTA_1.%X14 := FALSE;
	    END_IF;
	    
	    
	    IF "T_FECHO_EV4.1_HMI".Q AND "EV4.1_ABERTA" AND "EV4.1_FECHADA" THEN  //Avaria fim de curso de abertura
	        "Estados_HMI".ALARMES_LISTA_1.%X15 := TRUE;
	    ELSE
	        "Estados_HMI".ALARMES_LISTA_1.%X15 := FALSE;
	    END_IF;
	END_REGION
	REGION ALARME_V5.1
	    IF "T_ABERTURA_EV5.1_HMI".Q AND NOT "EV5.1_ABERTA" THEN  //Válvula não abriu
	        "Estados_HMI".ALARMES_LISTA_2.%X0 := TRUE;
	    ELSE
	        "Estados_HMI".ALARMES_LISTA_2.%X0 := FALSE;
	    END_IF;
	    
	    
	    IF "T_ABERTURA_EV5.1_HMI".Q AND "EV5.1_ABERTA" AND "EV5.1_FECHADA" THEN  //Avaria fim de curso de fecho
	        "Estados_HMI".ALARMES_LISTA_2.%X1 := TRUE;
	    ELSE
	        "Estados_HMI".ALARMES_LISTA_2.%X1 := FALSE;
	    END_IF;
	    
	    
	    IF "T_FECHO_EV5.1_HMI".Q AND NOT "EV5.1_FECHADA" THEN  //Válvula não fechou
	        "Estados_HMI".ALARMES_LISTA_2.%X2 := TRUE;
	    ELSE
	        "Estados_HMI".ALARMES_LISTA_2.%X2 := FALSE;
	    END_IF;
	    
	    
	    IF "T_FECHO_EV5.1_HMI".Q AND "EV5.1_ABERTA" AND "EV5.1_FECHADA" THEN  //Avaria fim de curso de abertura
	        "Estados_HMI".ALARMES_LISTA_2.%X3 := TRUE;
	    ELSE
	        "Estados_HMI".ALARMES_LISTA_2.%X3 := FALSE;
	    END_IF;
	END_REGION
	
	//Alarmes filtro 2
	//
	REGION ALARME_V1.2
	    IF "T_ABERTURA_EV1.2_HMI".Q AND NOT "EV1.2_ABERTA" THEN  //Válvula não abriu
	        "Estados_HMI".ALARMES_LISTA_2.%X4 := TRUE;
	    ELSE
	        "Estados_HMI".ALARMES_LISTA_2.%X4 := FALSE;
	    END_IF;
	    
	    
	    IF "T_ABERTURA_EV1.2_HMI".Q AND "EV1.2_ABERTA" AND "EV1.2_FECHADA" THEN  //Avaria fim de curso de fecho
	        "Estados_HMI".ALARMES_LISTA_2.%X5 := TRUE;
	    ELSE
	        "Estados_HMI".ALARMES_LISTA_2.%X5 := FALSE;
	    END_IF;
	    
	    
	    IF "T_FECHO_EV1.2_HMI".Q AND NOT "EV1.2_FECHADA" THEN  //Válvula não fechou
	        "Estados_HMI".ALARMES_LISTA_2.%X6 := TRUE;
	    ELSE
	        "Estados_HMI".ALARMES_LISTA_2.%X6 := FALSE;
	    END_IF;
	    
	    
	    IF "T_FECHO_EV1.2_HMI".Q AND "EV1.2_ABERTA" AND "EV1.2_FECHADA" THEN  //Avaria fim de curso de abertura
	        "Estados_HMI".ALARMES_LISTA_2.%X7 := TRUE;
	    ELSE
	        "Estados_HMI".ALARMES_LISTA_2.%X7 := FALSE;
	    END_IF;
	END_REGION
	REGION ALARME_V2.2
	    IF "T_ABERTURA_EV2.2_HMI".Q AND NOT "EV2.2_ABERTA" THEN  //Válvula não abriu
	        "Estados_HMI".ALARMES_LISTA_2.%X8 := TRUE;
	    ELSE
	        "Estados_HMI".ALARMES_LISTA_2.%X8 := FALSE;
	    END_IF;
	    
	    
	    IF "T_ABERTURA_EV2.2_HMI".Q AND "EV2.2_ABERTA" AND "EV2.2_FECHADA" THEN  //Avaria fim de curso de fecho
	        "Estados_HMI".ALARMES_LISTA_2.%X9 := TRUE;
	    ELSE
	        "Estados_HMI".ALARMES_LISTA_2.%X9 := FALSE;
	    END_IF;
	    
	    
	    IF "T_FECHO_EV2.2_HMI".Q AND NOT "EV2.2_FECHADA" THEN  //Válvula não fechou
	        "Estados_HMI".ALARMES_LISTA_2.%X10 := TRUE;
	    ELSE
	        "Estados_HMI".ALARMES_LISTA_2.%X10 := FALSE;
	    END_IF;
	    
	    
	    IF "T_FECHO_EV2.2_HMI".Q AND "EV2.2_ABERTA" AND "EV2.2_FECHADA" THEN  //Avaria fim de curso de abertura
	        "Estados_HMI".ALARMES_LISTA_2.%X11 := TRUE;
	    ELSE
	        "Estados_HMI".ALARMES_LISTA_2.%X11 := FALSE;
	    END_IF;
	END_REGION
	REGION ALARME_V3.2
	    IF "T_ABERTURA_EV3.2_HMI".Q AND NOT "EV3.2_ABERTA" THEN  //Válvula não abriu
	        "Estados_HMI".ALARMES_LISTA_2.%X12 := TRUE;
	    ELSE
	        "Estados_HMI".ALARMES_LISTA_2.%X12 := FALSE;
	    END_IF;
	    
	    
	    IF "T_ABERTURA_EV3.2_HMI".Q AND "EV3.2_ABERTA" AND "EV3.2_FECHADA" THEN  //Avaria fim de curso de fecho
	        "Estados_HMI".ALARMES_LISTA_2.%X13 := TRUE;
	    ELSE
	        "Estados_HMI".ALARMES_LISTA_2.%X13 := FALSE;
	    END_IF;
	    
	    
	    IF "T_FECHO_EV3.2_HMI".Q AND NOT "EV3.2_FECHADA" THEN  //Válvula não fechou
	        "Estados_HMI".ALARMES_LISTA_2.%X14 := TRUE;
	    ELSE
	        "Estados_HMI".ALARMES_LISTA_2.%X14 := FALSE;
	    END_IF;
	    
	    
	    IF "T_FECHO_EV3.2_HMI".Q AND "EV3.2_ABERTA" AND "EV3.2_FECHADA" THEN  //Avaria fim de curso de abertura
	        "Estados_HMI".ALARMES_LISTA_2.%X15 := TRUE;
	    ELSE
	        "Estados_HMI".ALARMES_LISTA_2.%X15 := FALSE;
	    END_IF;
	END_REGION
	REGION ALARME_V4.2
	    IF "T_ABERTURA_EV4.2_HMI".Q AND NOT "EV4.2_ABERTA" THEN  //Válvula não abriu
	        "Estados_HMI".ALARMES_LISTA_3.%X0 := TRUE;
	    ELSE
	        "Estados_HMI".ALARMES_LISTA_3.%X0 := FALSE;
	    END_IF;
	    
	    
	    IF "T_ABERTURA_EV4.2_HMI".Q AND "EV4.2_ABERTA" AND "EV4.2_FECHADA" THEN  //Avaria fim de curso de fecho
	        "Estados_HMI".ALARMES_LISTA_3.%X1 := TRUE;
	    ELSE
	        "Estados_HMI".ALARMES_LISTA_3.%X1 := FALSE;
	    END_IF;
	    
	    
	    IF "T_FECHO_EV4.2_HMI".Q AND NOT "EV4.2_FECHADA" THEN  //Válvula não fechou
	        "Estados_HMI".ALARMES_LISTA_3.%X2 := TRUE;
	    ELSE
	        "Estados_HMI".ALARMES_LISTA_3.%X2 := FALSE;
	    END_IF;
	    
	    
	    IF "T_FECHO_EV4.2_HMI".Q AND "EV4.2_ABERTA" AND "EV4.2_FECHADA" THEN  //Avaria fim de curso de abertura
	        "Estados_HMI".ALARMES_LISTA_3.%X3 := TRUE;
	    ELSE
	        "Estados_HMI".ALARMES_LISTA_3.%X3 := FALSE;
	    END_IF;
	END_REGION
	REGION ALARME_V5.2
	    IF "T_ABERTURA_EV5.2_HMI".Q AND NOT "EV5.2_ABERTA" THEN  //Válvula não abriu
	        "Estados_HMI".ALARMES_LISTA_3.%X4 := TRUE;
	    ELSE
	        "Estados_HMI".ALARMES_LISTA_3.%X4 := FALSE;
	    END_IF;
	    
	    
	    IF "T_ABERTURA_EV5.2_HMI".Q AND "EV5.2_ABERTA" AND "EV5.2_FECHADA" THEN  //Avaria fim de curso de fecho
	        "Estados_HMI".ALARMES_LISTA_3.%X5 := TRUE;
	    ELSE
	        "Estados_HMI".ALARMES_LISTA_3.%X5 := FALSE;
	    END_IF;
	    
	    
	    IF "T_FECHO_EV5.2_HMI".Q AND NOT "EV5.2_FECHADA" THEN  //Válvula não fechou
	        "Estados_HMI".ALARMES_LISTA_3.%X6 := TRUE;
	    ELSE
	        "Estados_HMI".ALARMES_LISTA_3.%X6 := FALSE;
	    END_IF;
	    
	    
	    IF "T_FECHO_EV5.2_HMI".Q AND "EV5.2_ABERTA" AND "EV5.2_FECHADA" THEN  //Avaria fim de curso de abertura
	        "Estados_HMI".ALARMES_LISTA_3.%X7 := TRUE;
	    ELSE
	        "Estados_HMI".ALARMES_LISTA_3.%X7 := FALSE;
	    END_IF;
	END_REGION
	
	//Alarmes Bombas
	//
	REGION ALARME_BOMBA_1
	    IF "AVARIA_BOMBA_1" = TRUE THEN
	        "Estados_HMI".ALARMES_LISTA_3.%X8 := TRUE;
	    ELSE
	        "Estados_HMI".ALARMES_LISTA_3.%X8 := FALSE;
	    END_IF;
	END_REGION
	
	REGION ALARME_BOMBA_2
	    IF "AVARIA_BOMBA_2" = TRUE THEN
	        "Estados_HMI".ALARMES_LISTA_3.%X9 := TRUE;
	    ELSE
	        "Estados_HMI".ALARMES_LISTA_3.%X9 := FALSE;
	    END_IF;
	END_REGION
	
	REGION ALARME_BOMBA_3
	    IF "AVARIA_BOMBA_3" = TRUE THEN
	        "Estados_HMI".ALARMES_LISTA_3.%X10 := TRUE;
	    ELSE
	        "Estados_HMI".ALARMES_LISTA_3.%X10 := FALSE;
	    END_IF;
	END_REGION
	
	
	
	
	
	
END_FUNCTION

FUNCTION "Estados_HMI" : Void
{ S7_Optimized_Access := 'TRUE' }
VERSION : 0.1

BEGIN
	"Estados_HMI_DB".MX201 := "MX201_ON";
	"Estados_HMI_DB".MX601 := "MX601_ON";
	"Estados_HMI_DB".XV101 := "XV101_ABERTA";
	
	IF "XV102_ABERTA" = TRUE
	THEN
	    "Estados_HMI_DB".XV102 := TRUE;
	END_IF;
	
	IF "XV102_FECHADA" = TRUE
	THEN
	    "Estados_HMI_DB".XV102 := FALSE;
	END_IF;
	
	"Estados_HMI_DB".BD601 := "BD601_ON";
	"Estados_HMI_DB".BD602 := "BD602_ON";
	"Estados_HMI_DB".BH201 := "BH201_ON";
	"Estados_HMI_DB".PH201 := "PH201_CONT_PH";
	"Estados_HMI_DB".RH201 := "RH201_CONT_REDOX";
	"Estados_HMI_DB".MX603 := "MX603_ON";
	"Estados_HMI_DB".BD603 := "BD603_ON";
	"Estados_HMI_DB".MX301 := "MX301_ON";
	"Estados_HMI_DB".PH301 := "PH301_CONT_PH";
	"Estados_HMI_DB".BM401 := "BM401_ON";
	"Estados_HMI_DB".MX604 := "MX604_ON";
	"Estados_HMI_DB".BD604 := "BD604_ON";
	"Estados_HMI_DB".MX605 := "MX605_ON";
	"Estados_HMI_DB".BD605 := "BD605_ON";
	"Estados_HMI_DB".BS001A := "BS001A_ON";
	"Estados_HMI_DB".BS001B := "BS001B_ON";
	"Estados_HMI_DB".BS501 := "BS501_ON";
END_FUNCTION

FUNCTION "Encrav_Inputs_HMI" : Void
{ S7_Optimized_Access := 'TRUE' }
VERSION : 0.1

BEGIN
	IF "Inputs_HMI".MAN_AUTO = TRUE THEN
	    "Inputs_HMI".ON_OFF_MX201 := FALSE;
	    "Inputs_HMI".ON_OFF_MX301 := FALSE;
	    "Inputs_HMI".ON_OFF_MX601 := FALSE;
	    "Inputs_HMI".ON_OFF_MX603 := FALSE;
	    "Inputs_HMI".ON_OFF_MX604 := FALSE;
	    "Inputs_HMI".ON_OFF_MX605 := FALSE;
	    "Inputs_HMI".ON_OFF_BS001A := FALSE;
	    "Inputs_HMI".ON_OFF_BS001B := FALSE;
	    "Inputs_HMI".ON_OFF_BS501 := FALSE;
	    "Inputs_HMI".ON_OFF_BH201 := FALSE;
	    "Inputs_HMI".ON_OFF_BM401 := FALSE;
	    "Inputs_HMI".ON_OFF_BD601 := FALSE;
	    "Inputs_HMI".ON_OFF_BD602 := FALSE;
	    "Inputs_HMI".ON_OFF_BD603 := FALSE;
	    "Inputs_HMI".ON_OFF_BD604 := FALSE;
	    "Inputs_HMI".ON_OFF_BD605 := FALSE;
	    "Inputs_HMI".ON_OFF_XV101 := FALSE;
	    "Inputs_HMI".ON_OFF_XV102 := FALSE;
	END_IF;
END_FUNCTION

FUNCTION "Estado_Ciclo_HMI" : Void
{ S7_Optimized_Access := 'TRUE' }
VERSION : 0.1

BEGIN
	IF ("Etapas_Grafcet_1".ETAPA_1 = TRUE) OR ("Inputs_HMI".MAN_AUTO = FALSE) OR ("BOT_EMERGÊNCIA" = FALSE) THEN
	    "Info_Ciclo".ESTADO_CICLO := FALSE;
	ELSE
	    "Info_Ciclo".ESTADO_CICLO := TRUE;
	END_IF;
END_FUNCTION

FUNCTION "Estado_Bombas" : Void
{ S7_Optimized_Access := 'TRUE' }
VERSION : 0.1

BEGIN
	//SINALIZAÇÃO DO ESTADO DAS BOMBAS PARA HMI
	
	REGION ESTADO_BOMBA_1
	    IF "BOMBA_1_VAR" = TRUE AND NOT "AVARIA_BOMBA_1" THEN  //BOMBA LIGADA
	        "Estados_HMI".BOMBA_1_ESTADO := 1;
	        "Estados_HMI".BOMBA_1_ESTADO_PAGCMD := 1;
	    END_IF;
	    
	    IF "BOMBA_1_VAR" = FALSE AND NOT "AVARIA_BOMBA_1" THEN  //BOMBA DESLIGADA
	        "Estados_HMI".BOMBA_1_ESTADO := 0;
	        "Estados_HMI".BOMBA_1_ESTADO_PAGCMD := 0;
	    END_IF;
	    
	    IF "AVARIA_BOMBA_1" THEN  //BOMBA AVARIA
	        "Estados_HMI".BOMBA_1_ESTADO := 2;
	        "Estados_HMI".BOMBA_1_ESTADO_PAGCMD := 2;
	    END_IF;
	END_REGION
	
	REGION ESTADO_BOMBA_2
	    IF "BOMBA_2_VAR" = TRUE AND NOT "AVARIA_BOMBA_2" THEN  //BOMBA LIGADA
	        "Estados_HMI".BOMBA_2_ESTADO := 1;
	        "Estados_HMI".BOMBA_2_ESTADO_PAGCMD := 1;
	    END_IF;
	    
	    IF "BOMBA_2_VAR" = FALSE AND NOT "AVARIA_BOMBA_2" THEN  //BOMBA DESLIGADA
	        "Estados_HMI".BOMBA_2_ESTADO := 0;
	        "Estados_HMI".BOMBA_2_ESTADO_PAGCMD := 0;
	    END_IF;
	    
	    IF "AVARIA_BOMBA_2" THEN  //BOMBA AVARIA
	        "Estados_HMI".BOMBA_2_ESTADO := 2;
	        "Estados_HMI".BOMBA_2_ESTADO_PAGCMD := 2;
	    END_IF;
	END_REGION
	
	REGION ESTADO_BOMBA_3
	    IF "BOMBA_3_RESERVA" = TRUE AND NOT "AVARIA_BOMBA_3" THEN  //BOMBA LIGADA
	        "Estados_HMI".BOMBA_3_ESTADO := 1;
	        "Estados_HMI".BOMBA_3_ESTADO_PAGCMD := 1;
	    END_IF;
	    
	    IF "BOMBA_3_RESERVA" = FALSE AND NOT "AVARIA_BOMBA_3" THEN  //BOMBA DESLIGADA
	        "Estados_HMI".BOMBA_3_ESTADO := 0;
	        "Estados_HMI".BOMBA_3_ESTADO_PAGCMD := 0;
	    END_IF;
	    
	    IF "AVARIA_BOMBA_3" THEN  //BOMBA AVARIA
	        "Estados_HMI".BOMBA_3_ESTADO := 2;
	        "Estados_HMI".BOMBA_3_ESTADO_PAGCMD := 2;
	    END_IF;
	END_REGION
END_FUNCTION

FUNCTION "Posição_EVs" : Void
{ S7_Optimized_Access := 'TRUE' }
VERSION : 0.1
   VAR_TEMP 
      "temp_clock_0.625Hz" : Int;
      "avaria_ev1.1" : Bool;
      "avaria_ev2.1" : Bool;
      "avaria_ev3.1" : Bool;
      "avaria_ev4.1" : Bool;
      "avaria_ev5.1" : Bool;
      "avaria_ev1.2" : Bool;
      "avaria_ev2.2" : Bool;
      "avaria_ev3.2" : Bool;
      "avaria_ev4.2" : Bool;
      "avaria_ev5.2" : Bool;
   END_VAR


BEGIN
	REGION POSICAO_FILTRO_1
	    IF "EV1.1_ABERTA" = TRUE AND "EV5.1_ABERTA" = TRUE AND
	        "EV2.1_FECHADA" = TRUE AND "EV4.1_FECHADA" = TRUE AND
	        "EV3.1_FECHADA" = TRUE AND
	        
	        "EV1.1_FECHADA" = FALSE AND "EV5.1_FECHADA" = FALSE AND
	        "EV2.1_ABERTA" = FALSE AND "EV4.1_ABERTA" = FALSE AND
	        "EV3.1_ABERTA" = FALSE
	    THEN
	        "Dados_Ciclo".POS_EVS_FILT_1 := 'FILTRACAO';
	    ELSE
	        
	        IF "EV2.1_ABERTA" = TRUE AND "EV3.1_ABERTA" = TRUE AND
	            "EV1.1_FECHADA" = TRUE AND "EV4.1_FECHADA" = TRUE AND
	            "EV5.1_FECHADA" = TRUE AND
	            
	            "EV2.1_FECHADA" = FALSE AND "EV3.1_FECHADA" = FALSE AND
	            "EV1.1_ABERTA" = FALSE AND "EV4.1_ABERTA" = FALSE AND
	            "EV5.1_ABERTA" = FALSE
	        THEN
	            "Dados_Ciclo".POS_EVS_FILT_1 := 'LAVAGEM';
	        ELSE
	            
	            IF "EV1.1_ABERTA" = TRUE AND "EV4.1_ABERTA" = TRUE AND
	                "EV2.1_FECHADA" = TRUE AND "EV3.1_FECHADA" = TRUE AND
	                "EV5.1_FECHADA" = TRUE AND
	                
	                "EV1.1_FECHADA" = FALSE AND "EV4.1_FECHADA" = FALSE AND
	                "EV2.1_ABERTA" = FALSE AND "EV3.1_ABERTA" = FALSE AND
	                "EV5.1_ABERTA" = FALSE
	            THEN
	                "Dados_Ciclo".POS_EVS_FILT_1 := 'RINSE';
	            ELSE
	                
	                IF "EV1.1_ABERTA" = TRUE AND "EV3.1_ABERTA" = TRUE AND
	                    "EV2.1_FECHADA" = TRUE AND "EV4.1_FECHADA" = TRUE AND
	                    "EV5.1_FECHADA" = TRUE AND
	                    
	                    "EV1.1_FECHADA" = FALSE AND "EV3.1_FECHADA" = FALSE AND
	                    "EV2.1_ABERTA" = FALSE AND "EV4.1_ABERTA" = FALSE AND
	                    "EV5.1_ABERTA" = FALSE
	                THEN
	                    "Dados_Ciclo".POS_EVS_FILT_1 := 'ESVAZIAMENTO';
	                ELSE
	                    
	                    IF "EV1.1_FECHADA" = TRUE AND "EV2.1_FECHADA" = TRUE AND
	                        "EV3.1_FECHADA" = TRUE AND "EV4.1_FECHADA" = TRUE AND
	                        "EV5.1_FECHADA" = TRUE AND
	                        
	                        "EV1.1_ABERTA" = FALSE AND "EV2.1_ABERTA" = FALSE AND
	                        "EV3.1_ABERTA" = FALSE AND "EV4.1_ABERTA" = FALSE AND
	                        "EV5.1_ABERTA" = FALSE
	                    THEN
	                        "Dados_Ciclo".POS_EVS_FILT_1 := 'FECHO';
	                    ELSE
	                        "Dados_Ciclo".POS_EVS_FILT_1 := 'NULL';
	                    END_IF;
	                END_IF;
	            END_IF;
	        END_IF;
	    END_IF;
	    
	END_REGION
	
	REGION POSICAO_FILTRO_2
	    IF "EV1.2_ABERTA" = TRUE AND "EV5.2_ABERTA" = TRUE AND
	        "EV2.2_FECHADA" = TRUE AND "EV4.2_FECHADA" = TRUE AND
	        "EV3.2_FECHADA" = TRUE AND
	        
	        "EV1.2_FECHADA" = FALSE AND "EV5.2_FECHADA" = FALSE AND
	        "EV2.2_ABERTA" = FALSE AND "EV4.2_ABERTA" = FALSE AND
	        "EV3.2_ABERTA" = FALSE
	    THEN
	        "Dados_Ciclo".POS_EVS_FILT_2 := 'FILTRACAO';
	    ELSE
	        
	        IF "EV2.2_ABERTA" = TRUE AND "EV3.2_ABERTA" = TRUE AND
	            "EV1.2_FECHADA" = TRUE AND "EV4.2_FECHADA" = TRUE AND
	            "EV5.2_FECHADA" = TRUE AND
	            
	            "EV2.2_FECHADA" = FALSE AND "EV3.2_FECHADA" = FALSE AND
	            "EV1.2_ABERTA" = FALSE AND "EV4.2_ABERTA" = FALSE AND
	            "EV5.2_ABERTA" = FALSE
	        THEN
	            "Dados_Ciclo".POS_EVS_FILT_2 := 'LAVAGEM';
	        ELSE
	            
	            IF "EV1.2_ABERTA" = TRUE AND "EV4.2_ABERTA" = TRUE AND
	                "EV2.2_FECHADA" = TRUE AND "EV3.2_FECHADA" = TRUE AND
	                "EV5.2_FECHADA" = TRUE AND
	                
	                "EV1.2_FECHADA" = FALSE AND "EV4.2_FECHADA" = FALSE AND
	                "EV2.2_ABERTA" = FALSE AND "EV3.2_ABERTA" = FALSE AND
	                "EV5.2_ABERTA" = FALSE
	            THEN
	                "Dados_Ciclo".POS_EVS_FILT_2 := 'RINSE';
	            ELSE
	                
	                IF "EV1.2_ABERTA" = TRUE AND "EV3.2_ABERTA" = TRUE AND
	                    "EV2.2_FECHADA" = TRUE AND "EV4.2_FECHADA" = TRUE AND
	                    "EV5.2_FECHADA" = TRUE AND
	                    
	                    "EV1.2_FECHADA" = FALSE AND "EV3.2_FECHADA" = FALSE AND
	                    "EV2.2_ABERTA" = FALSE AND "EV4.2_ABERTA" = FALSE AND
	                    "EV5.2_ABERTA" = FALSE
	                THEN
	                    "Dados_Ciclo".POS_EVS_FILT_2 := 'ESVAZIAMENTO';
	                ELSE
	                    
	                    IF "EV1.2_FECHADA" = TRUE AND "EV2.2_FECHADA" = TRUE AND
	                        "EV3.2_FECHADA" = TRUE AND "EV4.2_FECHADA" = TRUE AND
	                        "EV5.2_FECHADA" = TRUE AND
	                        
	                        "EV1.2_ABERTA" = FALSE AND "EV2.2_ABERTA" = FALSE AND
	                        "EV3.2_ABERTA" = FALSE AND "EV4.2_ABERTA" = FALSE AND
	                        "EV5.2_ABERTA" = FALSE
	                    THEN
	                        "Dados_Ciclo".POS_EVS_FILT_2 := 'FECHO';
	                    ELSE
	                        "Dados_Ciclo".POS_EVS_FILT_2 := 'NULL';
	                    END_IF;
	                END_IF;
	            END_IF;
	        END_IF;
	    END_IF;
	    
	END_REGION
	
	//Envio de estado de avaria para hmi
	//conversão de clock para piscar quando ocorre avaria de EVs
	#"temp_clock_0.625Hz" := BOOL_TO_INT("Clock_0.625Hz");
	
	//FILTRO 1
	REGION Estado_EV1.1
	    "T_ABERTURA_EV1.1_HMI".TON(IN := "EV1.1",                   //Quando EV1.1 recebe sinal para abrir, inicia uma contagem
	   PT := "Inputs_HMI".T_POS_EVS);
	    
	    "T_FECHO_EV1.1_HMI".TON(IN := NOT "EV1.1",                  //Quando EV1.1 recebe sinal para fechar, inicia uma contagem
	   PT := "Inputs_HMI".T_POS_EVS);
	                                                                //No final da contagem avalia se a EV está na posição pretendida
	                                                                
	    IF ("T_ABERTURA_EV1.1_HMI".Q AND (NOT "EV1.1_ABERTA" OR ("EV1.1_ABERTA" AND "EV1.1_FECHADA"))) OR   //Condição de avaria
	        ("T_FECHO_EV1.1_HMI".Q AND (NOT "EV1.1_FECHADA" OR ("EV1.1_ABERTA" AND "EV1.1_FECHADA"))) THEN  //para evitar dois estados 
	       #"avaria_ev1.1" := TRUE;                                                                     //na pagcmd evs da hmi
	    ELSE
	       #"avaria_ev1.1" := FALSE;
	    END_IF;
	    
	    
	    IF #"avaria_ev1.1" = FALSE AND "EV1.1_ABERTA" AND NOT "EV1.1_FECHADA" THEN //Condição de EV1.1 ABERTA
	        "Estados_HMI"."EV1.1_ESTADO" := 1;
	        "Estados_HMI"."EV1.1_ESTADO_PAGCMD" := 1;
	    END_IF;
	    
	    
	    IF #"avaria_ev1.1" = FALSE AND "EV1.1_FECHADA" AND NOT "EV1.1_ABERTA" THEN //Condição de EV1.1 Fechada
	        "Estados_HMI"."EV1.1_ESTADO" := 0;
	        "Estados_HMI"."EV1.1_ESTADO_PAGCMD" := 0;
	    END_IF;
	    
	    
	    IF ("T_ABERTURA_EV1.1_HMI".Q AND (NOT "EV1.1_ABERTA" OR ("EV1.1_ABERTA" AND "EV1.1_FECHADA"))) OR   //Condição de avaria
	        ("T_FECHO_EV1.1_HMI".Q AND (NOT "EV1.1_FECHADA" OR ("EV1.1_ABERTA" AND "EV1.1_FECHADA"))) THEN
	        
	        "Estados_HMI"."EV1.1_ESTADO_PAGCMD" := 2;
	        
	        CASE #"temp_clock_0.625Hz" OF
	            0:
	                "Estados_HMI"."EV1.1_ESTADO" := 0;
	                
	            1:
	                "Estados_HMI"."EV1.1_ESTADO" := 2;
	        END_CASE;
	    END_IF;
	    
	    IF "T_ABERTURA_EV1.1_HMI".Q = FALSE AND "T_FECHO_EV1.1_HMI".Q = FALSE AND
	        "EV1.1_ABERTA" = FALSE AND "EV1.1_FECHADA" = FALSE THEN  //Condição de transição das EVs
	        
	        "Estados_HMI"."EV1.1_ESTADO_PAGCMD" := 3;
	        
	        CASE #"temp_clock_0.625Hz" OF
	            0:
	                "Estados_HMI"."EV1.1_ESTADO" := 0;
	            1:
	                "Estados_HMI"."EV1.1_ESTADO" := 3;
	        END_CASE;
	    END_IF;
	    
	END_REGION
	
	REGION Estado_EV2.1
	    
	    "T_ABERTURA_EV2.1_HMI".TON(IN := "EV2.1",                   //Quando EV2.1 recebe sinal para abrir, inicia uma contagem
	                               PT := "Inputs_HMI".T_POS_EVS);
	    
	    "T_FECHO_EV2.1_HMI".TON(IN := NOT "EV2.1",                  //Quando EV2.1 recebe sinal para fechar, inicia uma contagem
	                            PT := "Inputs_HMI".T_POS_EVS);
	                                                                //No final da contagem avalia se a EV está na posição pretendida
	                                                                
	    IF ("T_ABERTURA_EV2.1_HMI".Q AND (NOT "EV2.1_ABERTA" OR ("EV2.1_ABERTA" AND "EV2.1_FECHADA"))) OR   //Condição de avaria
	        ("T_FECHO_EV2.1_HMI".Q AND (NOT "EV2.1_FECHADA" OR ("EV2.1_ABERTA" AND "EV2.1_FECHADA"))) THEN
	        #"avaria_ev2.1" := TRUE;
	    ELSE
	        #"avaria_ev2.1" := FALSE;
	    END_IF;
	    
	                                                                
	    IF #"avaria_ev2.1" = FALSE AND"EV2.1_ABERTA" AND NOT "EV2.1_FECHADA" THEN //Condição de EV2.1 ABERTA
	        "Estados_HMI"."EV2.1_ESTADO" := 1;
	        "Estados_HMI"."EV2.1_ESTADO_PAGCMD" := 1;
	    END_IF;
	    
	    
	    IF #"avaria_ev2.1" = FALSE AND"EV2.1_FECHADA" AND NOT "EV2.1_ABERTA" THEN //Condição de EV2.1 Fechada
	        "Estados_HMI"."EV2.1_ESTADO" := 0;
	        "Estados_HMI"."EV2.1_ESTADO_PAGCMD" := 0;
	    END_IF;
	    
	    
	    IF ("T_ABERTURA_EV2.1_HMI".Q AND (NOT "EV2.1_ABERTA" OR ("EV2.1_ABERTA" AND "EV2.1_FECHADA"))) OR   //Condição de avaria
	        ("T_FECHO_EV2.1_HMI".Q AND (NOT "EV2.1_FECHADA" OR ("EV2.1_ABERTA" AND "EV2.1_FECHADA"))) THEN
	        
	        "Estados_HMI"."EV2.1_ESTADO_PAGCMD" := 2;
	        
	        CASE #"temp_clock_0.625Hz" OF
	            0:
	                "Estados_HMI"."EV2.1_ESTADO" := 0;
	            1:
	                "Estados_HMI"."EV2.1_ESTADO" := 2;
	        END_CASE;
	    END_IF;
	    
	    IF "T_ABERTURA_EV2.1_HMI".Q = FALSE AND "T_FECHO_EV2.1_HMI".Q = FALSE AND
	        "EV2.1_ABERTA" = FALSE AND "EV2.1_FECHADA" = FALSE THEN  //Condição de transição das EVs
	        
	        "Estados_HMI"."EV2.1_ESTADO_PAGCMD" := 3;
	        
	        CASE #"temp_clock_0.625Hz" OF
	            0:
	                "Estados_HMI"."EV2.1_ESTADO" := 0;
	            1:
	                "Estados_HMI"."EV2.1_ESTADO" := 3;
	        END_CASE;
	    END_IF;
	                                                                
	END_REGION
	
	REGION Estado_EV3.1
	    
	    "T_ABERTURA_EV3.1_HMI".TON(IN := "EV3.1",                   //Quando EV3.1 recebe sinal para abrir, inicia uma contagem
	                               PT := "Inputs_HMI".T_POS_EVS);
	    
	    "T_FECHO_EV3.1_HMI".TON(IN := NOT "EV3.1",                  //Quando EV3.1 recebe sinal para fechar, inicia uma contagem
	                            PT := "Inputs_HMI".T_POS_EVS);
	    //No final da contagem avalia se a EV está na posição pretendida
	    
	    IF ("T_ABERTURA_EV3.1_HMI".Q AND (NOT "EV3.1_ABERTA" OR ("EV3.1_ABERTA" AND "EV3.1_FECHADA"))) OR   //Condição de avaria
	        ("T_FECHO_EV3.1_HMI".Q AND (NOT "EV3.1_FECHADA" OR ("EV3.1_ABERTA" AND "EV3.1_FECHADA"))) THEN
	        #"avaria_ev3.1" := TRUE;
	    ELSE
	        #"avaria_ev3.1" := FALSE;
	    END_IF;
	    
	    
	    IF #"avaria_ev3.1" = FALSE AND "EV3.1_ABERTA" AND NOT "EV3.1_FECHADA" THEN //Condição de EV3.1 ABERTA
	        "Estados_HMI"."EV3.1_ESTADO" := 1;
	        "Estados_HMI"."EV3.1_ESTADO_PAGCMD" := 1;
	    END_IF;
	    
	    
	    IF #"avaria_ev3.1" = FALSE AND "EV3.1_FECHADA" AND NOT "EV3.1_ABERTA" THEN //Condição de EV3.1 Fechada
	        "Estados_HMI"."EV3.1_ESTADO" := 0;
	        "Estados_HMI"."EV3.1_ESTADO_PAGCMD" := 0;
	    END_IF;
	    
	    
	    IF ("T_ABERTURA_EV3.1_HMI".Q AND (NOT "EV3.1_ABERTA" OR ("EV3.1_ABERTA" AND "EV3.1_FECHADA"))) OR   //Condição de avaria
	        ("T_FECHO_EV3.1_HMI".Q AND (NOT "EV3.1_FECHADA" OR ("EV3.1_ABERTA" AND "EV3.1_FECHADA"))) THEN
	        
	        "Estados_HMI"."EV3.1_ESTADO_PAGCMD" := 2;
	        
	        CASE #"temp_clock_0.625Hz" OF
	            0:
	                "Estados_HMI"."EV3.1_ESTADO" := 0;
	            1:
	                "Estados_HMI"."EV3.1_ESTADO" := 2;
	        END_CASE;
	    END_IF;
	    
	    IF "T_ABERTURA_EV3.1_HMI".Q = FALSE AND "T_FECHO_EV3.1_HMI".Q = FALSE AND
	        "EV3.1_ABERTA" = FALSE AND "EV3.1_FECHADA" = FALSE THEN  //Condição de transição das EVs
	        
	        "Estados_HMI"."EV3.1_ESTADO_PAGCMD" := 3;
	        
	        CASE #"temp_clock_0.625Hz" OF
	            0:
	                "Estados_HMI"."EV3.1_ESTADO" := 0;
	            1:
	                "Estados_HMI"."EV3.1_ESTADO" := 3;
	        END_CASE;
	    END_IF;
	    
	END_REGION
	
	REGION Estado_EV4.1
	    
	    "T_ABERTURA_EV4.1_HMI".TON(IN := "EV4.1",                   //Quando EV4.1 recebe sinal para abrir, inicia uma contagem
	                               PT := "Inputs_HMI".T_POS_EVS);
	    
	    "T_FECHO_EV4.1_HMI".TON(IN := NOT "EV4.1",                  //Quando EV4.1 recebe sinal para fechar, inicia uma contagem
	                            PT := "Inputs_HMI".T_POS_EVS);
	                                                                //No final da contagem avalia se a EV está na posição pretendida
	                                                                
	    IF ("T_ABERTURA_EV4.1_HMI".Q AND (NOT "EV4.1_ABERTA" OR ("EV4.1_ABERTA" AND "EV4.1_FECHADA"))) OR   //Condição de avaria
	        ("T_FECHO_EV4.1_HMI".Q AND (NOT "EV4.1_FECHADA" OR ("EV4.1_ABERTA" AND "EV4.1_FECHADA"))) THEN
	        #"avaria_ev4.1" := TRUE;
	    ELSE
	        #"avaria_ev4.1" := FALSE;
	    END_IF;
	                                                                
	    IF #"avaria_ev4.1" = FALSE AND "EV4.1_ABERTA" AND NOT "EV4.1_FECHADA" THEN //Condição de EV4.1 ABERTA
	        "Estados_HMI"."EV4.1_ESTADO" := 1;
	        "Estados_HMI"."EV4.1_ESTADO_PAGCMD" := 1;
	    END_IF;
	    
	    
	    IF #"avaria_ev4.1" = FALSE AND "EV4.1_FECHADA" AND NOT "EV4.1_ABERTA" THEN //Condição de EV4.1 Fechada
	        "Estados_HMI"."EV4.1_ESTADO" := 0;
	        "Estados_HMI"."EV4.1_ESTADO_PAGCMD" := 0;
	    END_IF;
	    
	    
	    IF ("T_ABERTURA_EV4.1_HMI".Q AND (NOT "EV4.1_ABERTA" OR ("EV4.1_ABERTA" AND "EV4.1_FECHADA"))) OR   //Condição de avaria
	        ("T_FECHO_EV4.1_HMI".Q AND (NOT "EV4.1_FECHADA" OR ("EV4.1_ABERTA" AND "EV4.1_FECHADA"))) THEN
	        
	        "Estados_HMI"."EV4.1_ESTADO_PAGCMD" := 2;
	        
	        CASE #"temp_clock_0.625Hz" OF
	            0:
	                "Estados_HMI"."EV4.1_ESTADO" := 0;
	            1:
	                "Estados_HMI"."EV4.1_ESTADO" := 2;
	        END_CASE;
	    END_IF;
	    
	    IF "T_ABERTURA_EV4.1_HMI".Q = FALSE AND "T_FECHO_EV4.1_HMI".Q = FALSE AND
	        "EV4.1_ABERTA" = FALSE AND "EV4.1_FECHADA" = FALSE THEN  //Condição de transição das EVs
	        
	        "Estados_HMI"."EV4.1_ESTADO_PAGCMD" := 3;
	        
	        CASE #"temp_clock_0.625Hz" OF
	            0:
	                "Estados_HMI"."EV4.1_ESTADO" := 0;
	            1:
	                "Estados_HMI"."EV4.1_ESTADO" := 3;
	        END_CASE;
	    END_IF;
	    
	END_REGION
	
	REGION Estado_EV5.1
	    
	    "T_ABERTURA_EV5.1_HMI".TON(IN := "EV5.1",                   //Quando EV5.1 recebe sinal para abrir, inicia uma contagem
	                               PT := "Inputs_HMI".T_POS_EVS);
	    
	    "T_FECHO_EV5.1_HMI".TON(IN := NOT "EV5.1",                  //Quando EV5.1 recebe sinal para fechar, inicia uma contagem
	                            PT := "Inputs_HMI".T_POS_EVS);
	                                                                //No final da contagem avalia se a EV está na posição pretendida
	                                                                
	    IF ("T_ABERTURA_EV5.1_HMI".Q AND (NOT "EV5.1_ABERTA" OR ("EV5.1_ABERTA" AND "EV5.1_FECHADA"))) OR   //Condição de avaria
	        ("T_FECHO_EV5.1_HMI".Q AND (NOT "EV5.1_FECHADA" OR ("EV5.1_ABERTA" AND "EV5.1_FECHADA"))) THEN
	        #"avaria_ev5.1" := TRUE;
	    ELSE
	        #"avaria_ev5.1" := FALSE;
	    END_IF;
	                                                                
	    IF #"avaria_ev5.1" = FALSE AND "EV5.1_ABERTA" AND NOT "EV5.1_FECHADA" THEN //Condição de EV5.1 ABERTA
	        "Estados_HMI"."EV5.1_ESTADO" := 1;
	        "Estados_HMI"."EV5.1_ESTADO_PAGCMD" := 1;
	    END_IF;
	    
	    
	    IF #"avaria_ev5.1" = FALSE AND "EV5.1_FECHADA" AND NOT "EV5.1_ABERTA" THEN //Condição de EV5.1 Fechada
	        "Estados_HMI"."EV5.1_ESTADO" := 0;
	        "Estados_HMI"."EV5.1_ESTADO_PAGCMD" := 0;
	    END_IF;
	    
	    
	    IF ("T_ABERTURA_EV5.1_HMI".Q AND (NOT "EV5.1_ABERTA" OR ("EV5.1_ABERTA" AND "EV5.1_FECHADA"))) OR   //Condição de avaria
	        ("T_FECHO_EV5.1_HMI".Q AND (NOT "EV5.1_FECHADA" OR ("EV5.1_ABERTA" AND "EV5.1_FECHADA"))) THEN
	        
	        "Estados_HMI"."EV5.1_ESTADO_PAGCMD" := 2;
	        
	        CASE #"temp_clock_0.625Hz" OF
	            0:
	                "Estados_HMI"."EV5.1_ESTADO" := 0;
	            1:
	                "Estados_HMI"."EV5.1_ESTADO" := 2;
	        END_CASE;
	    END_IF;
	    
	    IF "T_ABERTURA_EV5.1_HMI".Q = FALSE AND "T_FECHO_EV5.1_HMI".Q = FALSE AND
	        "EV5.1_ABERTA" = FALSE AND "EV5.1_FECHADA" = FALSE THEN  //Condição de transição das EVs
	        
	        "Estados_HMI"."EV5.1_ESTADO_PAGCMD" := 3;
	        
	        CASE #"temp_clock_0.625Hz" OF
	            0:
	                "Estados_HMI"."EV5.1_ESTADO" := 0;
	            1:
	                "Estados_HMI"."EV5.1_ESTADO" := 3;
	        END_CASE;
	    END_IF;
	    
	END_REGION
	
	//FILTRO 2
	
	REGION Estado_EV1.2
	    "T_ABERTURA_EV1.2_HMI".TON(IN := "EV1.2",                   //Quando EV1.2 recebe sinal para abrir, inicia uma contagem
	                               PT := "Inputs_HMI".T_POS_EVS);
	    
	    "T_FECHO_EV1.2_HMI".TON(IN := NOT "EV1.2",                  //Quando EV1.2 recebe sinal para fechar, inicia uma contagem
	                            PT := "Inputs_HMI".T_POS_EVS);
	    //No final da contagem avalia se a EV está na posição pretendida
	    
	    IF ("T_ABERTURA_EV1.2_HMI".Q AND (NOT "EV1.2_ABERTA" OR ("EV1.2_ABERTA" AND "EV1.2_FECHADA"))) OR   //Condição de avaria
	        ("T_FECHO_EV1.2_HMI".Q AND (NOT "EV1.2_FECHADA" OR ("EV1.2_ABERTA" AND "EV1.2_FECHADA"))) THEN
	        #"avaria_ev1.2" := TRUE;
	    ELSE
	        #"avaria_ev1.2" := FALSE;
	    END_IF;
	        
	    IF #"avaria_ev1.2" = FALSE AND "EV1.2_ABERTA" AND NOT "EV1.2_FECHADA" THEN //Condição de EV1.2 ABERTA
	        "Estados_HMI"."EV1.2_ESTADO" := 1;
	        "Estados_HMI"."EV1.2_ESTADO_PAGCMD" := 1;
	    END_IF;
	    
	    
	    IF #"avaria_ev1.2" = FALSE AND "EV1.2_FECHADA" AND NOT "EV1.2_ABERTA" THEN //Condição de EV1.2 Fechada
	        "Estados_HMI"."EV1.2_ESTADO" := 0;
	        "Estados_HMI"."EV1.2_ESTADO_PAGCMD" := 0;
	    END_IF;
	    
	    
	    IF ("T_ABERTURA_EV1.2_HMI".Q AND (NOT "EV1.2_ABERTA" OR ("EV1.2_ABERTA" AND "EV1.2_FECHADA"))) OR   //Condição de avaria
	        ("T_FECHO_EV1.2_HMI".Q AND (NOT "EV1.2_FECHADA" OR ("EV1.2_ABERTA" AND "EV1.2_FECHADA"))) THEN
	        
	        "Estados_HMI"."EV1.2_ESTADO_PAGCMD" := 2;
	        
	        CASE #"temp_clock_0.625Hz" OF
	            0:
	                "Estados_HMI"."EV1.2_ESTADO" := 0;
	            1:
	                "Estados_HMI"."EV1.2_ESTADO" := 2;
	        END_CASE;
	    END_IF;
	    
	    IF "T_ABERTURA_EV1.2_HMI".Q = FALSE AND "T_FECHO_EV1.2_HMI".Q = FALSE AND
	        "EV1.2_ABERTA" = FALSE AND "EV1.2_FECHADA" = FALSE THEN  //Condição de transição das EVs
	        
	        "Estados_HMI"."EV1.2_ESTADO_PAGCMD" := 3;
	        
	        CASE #"temp_clock_0.625Hz" OF
	            0:
	                "Estados_HMI"."EV1.2_ESTADO" := 0;
	            1:
	                "Estados_HMI"."EV1.2_ESTADO" := 3;
	        END_CASE;
	    END_IF;
	    
	END_REGION
	
	REGION Estado_EV2.2
	    
	    "T_ABERTURA_EV2.2_HMI".TON(IN := "EV2.2",                   //Quando EV2.2 recebe sinal para abrir, inicia uma contagem
	                               PT := "Inputs_HMI".T_POS_EVS);
	    
	    "T_FECHO_EV2.2_HMI".TON(IN := NOT "EV2.2",                  //Quando EV2.2 recebe sinal para fechar, inicia uma contagem
	                            PT := "Inputs_HMI".T_POS_EVS);
	    //No final da contagem avalia se a EV está na posição pretendida
	    
	    IF ("T_ABERTURA_EV2.2_HMI".Q AND (NOT "EV2.2_ABERTA" OR ("EV2.2_ABERTA" AND "EV2.2_FECHADA"))) OR   //Condição de avaria
	        ("T_FECHO_EV2.2_HMI".Q AND (NOT "EV2.2_FECHADA" OR ("EV2.2_ABERTA" AND "EV2.2_FECHADA"))) THEN
	        #"avaria_ev2.2" := TRUE;
	    ELSE
	        #"avaria_ev2.2" := FALSE;
	    END_IF;
	    
	    IF #"avaria_ev2.2" = FALSE AND "EV2.2_ABERTA" AND NOT "EV2.2_FECHADA" THEN //Condição de EV2.2 ABERTA
	        "Estados_HMI"."EV2.2_ESTADO" := 1;
	        "Estados_HMI"."EV2.2_ESTADO_PAGCMD" := 1;
	    END_IF;
	    
	    
	    IF #"avaria_ev2.2" = FALSE AND "EV2.2_FECHADA" AND NOT "EV2.2_ABERTA" THEN //Condição de EV2.2 Fechada
	        "Estados_HMI"."EV2.2_ESTADO" := 0;
	        "Estados_HMI"."EV2.2_ESTADO_PAGCMD" := 0;
	    END_IF;
	    
	    
	    IF ("T_ABERTURA_EV2.2_HMI".Q AND (NOT "EV2.2_ABERTA" OR ("EV2.2_ABERTA" AND "EV2.2_FECHADA"))) OR   //Condição de avaria
	        ("T_FECHO_EV2.2_HMI".Q AND (NOT "EV2.2_FECHADA" OR ("EV2.2_ABERTA" AND "EV2.2_FECHADA"))) THEN
	        
	        "Estados_HMI"."EV2.2_ESTADO_PAGCMD" := 2;
	        
	        CASE #"temp_clock_0.625Hz" OF
	            0:
	                "Estados_HMI"."EV2.2_ESTADO" := 0;
	            1:
	                "Estados_HMI"."EV2.2_ESTADO" := 2;
	        END_CASE;
	    END_IF;
	    
	    IF "T_ABERTURA_EV2.2_HMI".Q = FALSE AND "T_FECHO_EV2.2_HMI".Q = FALSE AND
	        "EV2.2_ABERTA" = FALSE AND "EV2.2_FECHADA" = FALSE THEN  //Condição de transição das EVs
	        
	        "Estados_HMI"."EV2.2_ESTADO_PAGCMD" := 3;
	        
	        CASE #"temp_clock_0.625Hz" OF
	            0:
	                "Estados_HMI"."EV2.2_ESTADO" := 0;
	            1:
	                "Estados_HMI"."EV2.2_ESTADO" := 3;
	        END_CASE;
	    END_IF;
	    
	END_REGION
	
	REGION Estado_EV3.2
	    
	    "T_ABERTURA_EV3.2_HMI".TON(IN := "EV3.2",                   //Quando EV3.2 recebe sinal para abrir, inicia uma contagem
	                               PT := "Inputs_HMI".T_POS_EVS);
	    
	    "T_FECHO_EV3.2_HMI".TON(IN := NOT "EV3.2",                  //Quando EV3.2 recebe sinal para fechar, inicia uma contagem
	                            PT := "Inputs_HMI".T_POS_EVS);
	    //No final da contagem avalia se a EV está na posição pretendida
	    
	    IF ("T_ABERTURA_EV3.2_HMI".Q AND (NOT "EV3.2_ABERTA" OR ("EV3.2_ABERTA" AND "EV3.2_FECHADA"))) OR   //Condição de avaria
	        ("T_FECHO_EV3.2_HMI".Q AND (NOT "EV3.2_FECHADA" OR ("EV3.2_ABERTA" AND "EV3.2_FECHADA"))) THEN
	        #"avaria_ev3.2" := TRUE;
	    ELSE
	        #"avaria_ev3.2" := FALSE;
	    END_IF;
	        
	    
	    IF #"avaria_ev3.2" = FALSE AND "EV3.2_ABERTA" AND NOT "EV3.2_FECHADA" THEN //Condição de EV3.2 ABERTA
	        "Estados_HMI"."EV3.2_ESTADO" := 1;
	        "Estados_HMI"."EV3.2_ESTADO_PAGCMD" := 1;
	    END_IF;
	    
	    
	    IF #"avaria_ev3.2" = FALSE AND "EV3.2_FECHADA" AND NOT "EV3.2_ABERTA" THEN //Condição de EV3.2 Fechada
	        "Estados_HMI"."EV3.2_ESTADO" := 0;
	        "Estados_HMI"."EV3.2_ESTADO_PAGCMD" := 0;
	    END_IF;
	    
	    
	    IF ("T_ABERTURA_EV3.2_HMI".Q AND (NOT "EV3.2_ABERTA" OR ("EV3.2_ABERTA" AND "EV3.2_FECHADA"))) OR   //Condição de avaria
	        ("T_FECHO_EV3.2_HMI".Q AND (NOT "EV3.2_FECHADA" OR ("EV3.2_ABERTA" AND "EV3.2_FECHADA"))) THEN
	        
	        "Estados_HMI"."EV3.2_ESTADO_PAGCMD" := 2;
	        
	        CASE #"temp_clock_0.625Hz" OF
	            0:
	                "Estados_HMI"."EV3.2_ESTADO" := 0;
	            1:
	                "Estados_HMI"."EV3.2_ESTADO" := 2;
	        END_CASE;
	    END_IF;
	    
	    IF "T_ABERTURA_EV3.2_HMI".Q = FALSE AND "T_FECHO_EV3.2_HMI".Q = FALSE AND
	        "EV3.2_ABERTA" = FALSE AND "EV3.2_FECHADA" = FALSE THEN  //Condição de transição das EVs
	        
	        "Estados_HMI"."EV3.2_ESTADO_PAGCMD" := 3;
	        
	        CASE #"temp_clock_0.625Hz" OF
	            0:
	                "Estados_HMI"."EV3.2_ESTADO" := 0;
	            1:
	                "Estados_HMI"."EV3.2_ESTADO" := 3;
	        END_CASE;
	    END_IF;
	    
	END_REGION
	
	REGION Estado_EV4.2
	    
	    "T_ABERTURA_EV4.2_HMI".TON(IN := "EV4.2",                   //Quando EV4.2 recebe sinal para abrir, inicia uma contagem
	                               PT := "Inputs_HMI".T_POS_EVS);
	    
	    "T_FECHO_EV4.2_HMI".TON(IN := NOT "EV4.2",                  //Quando EV4.2 recebe sinal para fechar, inicia uma contagem
	                            PT := "Inputs_HMI".T_POS_EVS);
	    //No final da contagem avalia se a EV está na posição pretendida
	    
	    IF ("T_ABERTURA_EV4.2_HMI".Q AND (NOT "EV4.2_ABERTA" OR ("EV4.2_ABERTA" AND "EV4.2_FECHADA"))) OR   //Condição de avaria
	        ("T_FECHO_EV4.2_HMI".Q AND (NOT "EV4.2_FECHADA" OR ("EV4.2_ABERTA" AND "EV4.2_FECHADA"))) THEN
	        #"avaria_ev4.2" := TRUE;
	    ELSE
	        #"avaria_ev4.2" := FALSE;
	    END_IF;
	    
	    
	    IF #"avaria_ev4.2" = FALSE AND "EV4.2_ABERTA" AND NOT "EV4.2_FECHADA" THEN //Condição de EV4.2 ABERTA
	        "Estados_HMI"."EV4.2_ESTADO" := 1;
	        "Estados_HMI"."EV4.2_ESTADO_PAGCMD" := 1;
	    END_IF;
	    
	    
	    IF #"avaria_ev4.2" = FALSE AND "EV4.2_FECHADA" AND NOT "EV4.2_ABERTA" THEN //Condição de EV4.2 Fechada
	        "Estados_HMI"."EV4.2_ESTADO" := 0;
	        "Estados_HMI"."EV4.2_ESTADO_PAGCMD" := 0;
	    END_IF;
	    
	    
	    IF ("T_ABERTURA_EV4.2_HMI".Q AND (NOT "EV4.2_ABERTA" OR ("EV4.2_ABERTA" AND "EV4.2_FECHADA"))) OR   //Condição de avaria
	        ("T_FECHO_EV4.2_HMI".Q AND (NOT "EV4.2_FECHADA" OR ("EV4.2_ABERTA" AND "EV4.2_FECHADA"))) THEN
	        
	        "Estados_HMI"."EV4.2_ESTADO_PAGCMD" := 2;
	        
	        CASE #"temp_clock_0.625Hz" OF
	            0:
	                "Estados_HMI"."EV4.2_ESTADO" := 0;
	            1:
	                "Estados_HMI"."EV4.2_ESTADO" := 2;
	        END_CASE;
	    END_IF;
	    
	    IF "T_ABERTURA_EV4.2_HMI".Q = FALSE AND "T_FECHO_EV4.2_HMI".Q = FALSE AND
	        "EV4.2_ABERTA" = FALSE AND "EV4.2_FECHADA" = FALSE THEN  //Condição de transição das EVs
	        
	        "Estados_HMI"."EV4.2_ESTADO_PAGCMD" := 3;
	        
	        CASE #"temp_clock_0.625Hz" OF
	            0:
	                "Estados_HMI"."EV4.2_ESTADO" := 0;
	            1:
	                "Estados_HMI"."EV4.2_ESTADO" := 3;
	        END_CASE;
	    END_IF;
	    
	END_REGION
	
	REGION Estado_EV5.2
	    
	    "T_ABERTURA_EV5.2_HMI".TON(IN := "EV5.2",                   //Quando EV5.2 recebe sinal para abrir, inicia uma contagem
	                               PT := "Inputs_HMI".T_POS_EVS);
	    
	    "T_FECHO_EV5.2_HMI".TON(IN := NOT "EV5.2",                  //Quando EV5.2 recebe sinal para fechar, inicia uma contagem
	                            PT := "Inputs_HMI".T_POS_EVS);
	    //No final da contagem avalia se a EV está na posição pretendida
	    
	    IF ("T_ABERTURA_EV5.2_HMI".Q AND (NOT "EV5.2_ABERTA" OR ("EV5.2_ABERTA" AND "EV5.2_FECHADA"))) OR   //Condição de avaria
	        ("T_FECHO_EV5.2_HMI".Q AND (NOT "EV5.2_FECHADA" OR ("EV5.2_ABERTA" AND "EV5.2_FECHADA"))) THEN
	        #"avaria_ev5.2" := TRUE;
	    ELSE
	        #"avaria_ev5.2" := FALSE;
	    END_IF;
	    
	    
	    IF #"avaria_ev5.2" = FALSE AND "EV5.2_ABERTA" AND NOT "EV5.2_FECHADA" THEN //Condição de EV5.2 ABERTA
	        "Estados_HMI"."EV5.2_ESTADO" := 1;
	        "Estados_HMI"."EV5.2_ESTADO_PAGCMD" := 1;
	    END_IF;
	    
	    
	    IF #"avaria_ev5.2" = FALSE AND "EV5.2_FECHADA" AND NOT "EV5.2_ABERTA" THEN //Condição de EV5.2 Fechada
	        "Estados_HMI"."EV5.2_ESTADO" := 0;
	        "Estados_HMI"."EV5.2_ESTADO_PAGCMD" := 0;
	    END_IF;
	    
	    
	    IF ("T_ABERTURA_EV5.2_HMI".Q AND (NOT "EV5.2_ABERTA" OR ("EV5.2_ABERTA" AND "EV5.2_FECHADA"))) OR   //Condição de avaria
	        ("T_FECHO_EV5.2_HMI".Q AND (NOT "EV5.2_FECHADA" OR ("EV5.2_ABERTA" AND "EV5.2_FECHADA"))) THEN
	        
	        "Estados_HMI"."EV5.2_ESTADO_PAGCMD" := 2;
	        
	        CASE #"temp_clock_0.625Hz" OF
	            0:
	                "Estados_HMI"."EV5.2_ESTADO" := 0;
	            1:
	                "Estados_HMI"."EV5.2_ESTADO" := 2;
	        END_CASE;
	    END_IF;
	    
	    IF "T_ABERTURA_EV5.2_HMI".Q = FALSE AND "T_FECHO_EV5.2_HMI".Q = FALSE AND
	        "EV5.2_ABERTA" = FALSE AND "EV5.2_FECHADA" = FALSE THEN  //Condição de transição das EVs
	        
	        "Estados_HMI"."EV5.2_ESTADO_PAGCMD" := 3;
	        
	        CASE #"temp_clock_0.625Hz" OF
	            0:
	                "Estados_HMI"."EV5.2_ESTADO" := 0;
	            1:
	                "Estados_HMI"."EV5.2_ESTADO" := 3;
	        END_CASE;
	    END_IF;
	    
	END_REGION
END_FUNCTION

FUNCTION "Conversão_TLAV_TRINSE" : Void
{ S7_Optimized_Access := 'TRUE' }
VERSION : 0.1

BEGIN
	//Conversão do tempo decorrido de lavagem e enxaguamento para minutos
	
	"Estados_HMI".T_LAV_MINUTOS := (TIME_TO_DINT("T_LAVAGEM".ET) MOD 3600000) / 60000;
	"Estados_HMI".T_RINSE_MINUTOS := (TIME_TO_DINT("T_RINSE".ET) MOD 3600000) / 60000;
END_FUNCTION

FUNCTION "Conversão_Tempo_Bombas" : Void
{ S7_Optimized_Access := 'TRUE' }
VERSION : 0.1
   VAR_TEMP 
      decimal_b2 : Real;
      result_b2 : Real;
      decimal_b3 : Real;
      result_b3 : Real;
      decimal_TON : Real;
      decimal_TOFF : Real;
      result_TON : Real;
      result_TOFF : Real;
   END_VAR


BEGIN
	//Conversão do tempo de alternancia das bombas introduzido na hmi (ex: em vez de introduzir 1.5 para dar 1h30m,
	//introduz-se 1.3 para da 1h30m
	
	
	//conversão T_ALTERNANCIA bombas 
	//
	#decimal_TON := ("Inputs_HMI".T_ALTERNANCIA_BOMBAS - TRUNC("Inputs_HMI".T_ALTERNANCIA_BOMBAS)) * 1.6667;
	#result_TON := TRUNC("Inputs_HMI".T_ALTERNANCIA_BOMBAS) + #decimal_TON;
	
	"Dados_Bombas".CONV_T_ALTERNANCIA_BOMBAS :=
	DINT_TO_TIME(
	             REAL_TO_DINT(#result_TON * 3600000));
	
	
	REGION leitura_tempos_func_bombas_para_hmi
	    
	    
	    "Dados_Bombas".HORAS_TON_B1 := "CNT_FUNC_B1".CV;
	    
	    "Dados_Bombas".HORAS_TON_B2 := "CNT_FUNC_B2".CV;
	    
	    "Dados_Bombas".HORAS_TON_B3 := "CNT_FUNC_B3".CV;
	   
	END_REGION
	
END_FUNCTION

FUNCTION "Controlo_Ciclo_Manual" : Void
{ S7_Optimized_Access := 'TRUE' }
VERSION : 0.1

BEGIN
	REGION controlo_etapa_anterior
	    //este bloco serve para saber qual a posição das válvulas antes da passagem para modo manual
	    IF "Etapas_Grafcet".ETAPA_1 = TRUE THEN
	        "Dados_Ciclo".ETAPA_ANTERIOR := 1;
	    END_IF;
	    
	    IF "Etapas_Grafcet".ETAPA_2 = TRUE THEN
	        "Dados_Ciclo".ETAPA_ANTERIOR := 2;
	    END_IF;
	    
	    IF "Etapas_Grafcet".ETAPA_3 = TRUE THEN
	        "Dados_Ciclo".ETAPA_ANTERIOR := 3;
	    END_IF;
	    
	    IF "Etapas_Grafcet".ETAPA_4 = TRUE THEN
	        "Dados_Ciclo".ETAPA_ANTERIOR := 4;
	    END_IF;
	    
	    IF "Etapas_Grafcet".ETAPA_5 = TRUE THEN
	        "Dados_Ciclo".ETAPA_ANTERIOR := 5;
	    END_IF;
	    
	    IF "Etapas_Grafcet".ETAPA_6 = TRUE THEN
	        "Dados_Ciclo".ETAPA_ANTERIOR := 6;
	    END_IF;
	    
	    IF "Etapas_Grafcet".ETAPA_7 = TRUE THEN
	        "Dados_Ciclo".ETAPA_ANTERIOR := 7;
	    END_IF;
	    
	    IF "Etapas_Grafcet".ETAPA_8 = TRUE THEN
	        "Dados_Ciclo".ETAPA_ANTERIOR := 8;
	    END_IF;
	    
	    IF "Etapas_Grafcet".ETAPA_9 = TRUE THEN
	        "Dados_Ciclo".ETAPA_ANTERIOR := 9;
	    END_IF;
	    
	END_REGION
	REGION controlo_etapa_13
	    // este bloco serve para reduzir o numero de contactos na nw13 do ciclo de limpeza
	    IF "Etapas_Grafcet".ETAPA_1 = TRUE OR
	       "Etapas_Grafcet".ETAPA_2 = TRUE OR
	       "Etapas_Grafcet".ETAPA_3 = TRUE OR
	       "Etapas_Grafcet".ETAPA_4 = TRUE OR
	       "Etapas_Grafcet".ETAPA_5 = TRUE OR
	       "Etapas_Grafcet".ETAPA_6 = TRUE OR
	       "Etapas_Grafcet".ETAPA_7 = TRUE OR
	       "Etapas_Grafcet".ETAPA_8 = TRUE OR
	       "Etapas_Grafcet".ETAPA_9 = TRUE
	    THEN
	        "Dados_Ciclo".ETAPA_N := TRUE;
	    END_IF;
	    
	    //reset às etaps de 1 a 9 pela etapa 13
	    IF "Etapas_Grafcet".ETAPA_13 = TRUE
	    THEN
	        "Etapas_Grafcet".ETAPA_1 := FALSE;
	        "Etapas_Grafcet".ETAPA_2 := FALSE;
	        "Etapas_Grafcet".ETAPA_3 := FALSE;
	        "Etapas_Grafcet".ETAPA_4 := FALSE;
	        "Etapas_Grafcet".ETAPA_5 := FALSE;
	        "Etapas_Grafcet".ETAPA_6 := FALSE;
	        "Etapas_Grafcet".ETAPA_7 := FALSE;
	        "Etapas_Grafcet".ETAPA_8 := FALSE;
	        "Etapas_Grafcet".ETAPA_9 := FALSE;
	        
	        "Dados_Ciclo".ETAPA_N := FALSE;
	    END_IF;
	    
	END_REGION
END_FUNCTION

DATA_BLOCK "Modbus_DB"   // DB28
VERSION : 0.1
// stored: AutoNumber false, InstanceOfName Modbus, InstanceOfType FB
"Modbus"
BEGIN
END_DATA_BLOCK

DATA_BLOCK "U241_Process_Data"   // DB213
VERSION : 0.1
// stored: AutoNumber false, InstanceOfName Inverter_Process_Data, InstanceOfType FB
"Inverter_Process_Data"
BEGIN
END_DATA_BLOCK

DATA_BLOCK "Centrador_Paletes_DB"   // DB11
VERSION : 0.1
// stored: AutoNumber true, InstanceOfName Centrador_Paletes, InstanceOfType FB
"Centrador_Paletes"
BEGIN
END_DATA_BLOCK

DATA_BLOCK "SINA_SPEED_Motor_Centrador_DB"   // DB11
AUTHOR : DRVDPS7
FAMILY : DRIVES
NAME : SINA_SPD
VERSION : 5.1
// stored: AutoNumber true, InstanceOfName SINA_SPEED_Motor_Centrador, InstanceOfType FB
"SINA_SPEED_Motor_Centrador"
BEGIN
END_DATA_BLOCK

DATA_BLOCK "U201_Process_Data"   // DB211
VERSION : 0.1
// stored: AutoNumber false, InstanceOfName Inverter_Process_Data, InstanceOfType FB
"Inverter_Process_Data"
BEGIN
END_DATA_BLOCK

DATA_BLOCK "U221_Process_Data"   // DB212
VERSION : 0.1
// stored: AutoNumber false, InstanceOfName Inverter_Process_Data, InstanceOfType FB
"Inverter_Process_Data"
BEGIN
END_DATA_BLOCK

DATA_BLOCK "CONTADOR_CICLOS"   // DB25
{ S7_Optimized_Access := 'TRUE' }
// stored: AutoNumber true, InstanceOfName IEC_COUNTER, OfSystemLibElement IEC_COUNTER, OfSystemLibVersion 1.0
"IEC_COUNTER"
   // VAR RETAIN
   //    CU : Bool;
   //    CD : Bool;
   //    R : Bool;
   //    LD : Bool;
   //    QU : Bool;
   //    QD : Bool;
   //    PV : Int;
   //    CV : Int;
   // END_VAR
BEGIN
END_DATA_BLOCK

DATA_BLOCK "ESTAB_NÍVEL_LSH101"   // DB17
{ S7_Optimized_Access := 'TRUE' }
// stored: AutoNumber true, InstanceOfName IEC_TIMER, OfSystemLibElement IEC_TIMER, OfSystemLibVersion 1.0
"IEC_TIMER"
   // VAR
   //    PT : Time;
   //    ET { ExternalWritable := 'False'} : Time;
   //    IN : Bool;
   //    Q { ExternalWritable := 'False'} : Bool;
   // END_VAR
BEGIN
END_DATA_BLOCK

DATA_BLOCK "ESTAB_NÍVEL_LSH201"   // DB21
{ S7_Optimized_Access := 'TRUE' }
// stored: AutoNumber true, InstanceOfName IEC_TIMER, OfSystemLibElement IEC_TIMER, OfSystemLibVersion 1.0
"IEC_TIMER"
   // VAR
   //    PT : Time;
   //    ET { ExternalWritable := 'False'} : Time;
   //    IN : Bool;
   //    Q { ExternalWritable := 'False'} : Bool;
   // END_VAR
BEGIN
END_DATA_BLOCK

DATA_BLOCK "ESTAB_NÍVEL_LSH301"   // DB23
{ S7_Optimized_Access := 'TRUE' }
// stored: AutoNumber true, InstanceOfName IEC_TIMER, OfSystemLibElement IEC_TIMER, OfSystemLibVersion 1.0
"IEC_TIMER"
   // VAR
   //    PT : Time;
   //    ET { ExternalWritable := 'False'} : Time;
   //    IN : Bool;
   //    Q { ExternalWritable := 'False'} : Bool;
   // END_VAR
BEGIN
END_DATA_BLOCK

DATA_BLOCK "ESTAB_NÍVEL_LSL001"   // DB19
{ S7_Optimized_Access := 'TRUE' }
// stored: AutoNumber true, InstanceOfName IEC_TIMER, OfSystemLibElement IEC_TIMER, OfSystemLibVersion 1.0
"IEC_TIMER"
   // VAR
   //    PT : Time;
   //    ET { ExternalWritable := 'False'} : Time;
   //    IN : Bool;
   //    Q { ExternalWritable := 'False'} : Bool;
   // END_VAR
BEGIN
END_DATA_BLOCK

DATA_BLOCK "ESTAB_NÍVEL_LSL101"   // DB20
{ S7_Optimized_Access := 'TRUE' }
// stored: AutoNumber true, InstanceOfName IEC_TIMER, OfSystemLibElement IEC_TIMER, OfSystemLibVersion 1.0
"IEC_TIMER"
   // VAR
   //    PT : Time;
   //    ET { ExternalWritable := 'False'} : Time;
   //    IN : Bool;
   //    Q { ExternalWritable := 'False'} : Bool;
   // END_VAR
BEGIN
END_DATA_BLOCK

DATA_BLOCK "ESTAB_NÍVEL_LSL201"   // DB22
{ S7_Optimized_Access := 'TRUE' }
// stored: AutoNumber true, InstanceOfName IEC_TIMER, OfSystemLibElement IEC_TIMER, OfSystemLibVersion 1.0
"IEC_TIMER"
   // VAR
   //    PT : Time;
   //    ET { ExternalWritable := 'False'} : Time;
   //    IN : Bool;
   //    Q { ExternalWritable := 'False'} : Bool;
   // END_VAR
BEGIN
END_DATA_BLOCK

DATA_BLOCK "ESTAB_NÍVEL_LSL301"   // DB24
{ S7_Optimized_Access := 'TRUE' }
// stored: AutoNumber true, InstanceOfName IEC_TIMER, OfSystemLibElement IEC_TIMER, OfSystemLibVersion 1.0
"IEC_TIMER"
   // VAR
   //    PT : Time;
   //    ET { ExternalWritable := 'False'} : Time;
   //    IN : Bool;
   //    Q { ExternalWritable := 'False'} : Bool;
   // END_VAR
BEGIN
END_DATA_BLOCK

DATA_BLOCK "ESTAB_NÍVEL_LSL501"   // DB18
{ S7_Optimized_Access := 'TRUE' }
// stored: AutoNumber true, InstanceOfName IEC_TIMER, OfSystemLibElement IEC_TIMER, OfSystemLibVersion 1.0
"IEC_TIMER"
   // VAR
   //    PT : Time;
   //    ET { ExternalWritable := 'False'} : Time;
   //    IN : Bool;
   //    Q { ExternalWritable := 'False'} : Bool;
   // END_VAR
BEGIN
END_DATA_BLOCK

DATA_BLOCK "TM0"   // DB5
{ S7_Optimized_Access := 'TRUE' }
// stored: AutoNumber true, InstanceOfName IEC_TIMER, OfSystemLibElement IEC_TIMER, OfSystemLibVersion 1.0
"IEC_TIMER"
   // VAR
   //    PT : Time;
   //    ET { ExternalWritable := 'False'} : Time;
   //    IN : Bool;
   //    Q { ExternalWritable := 'False'} : Bool;
   // END_VAR
BEGIN
END_DATA_BLOCK

DATA_BLOCK "TM1"   // DB6
{ S7_Optimized_Access := 'TRUE' }
// stored: AutoNumber true, InstanceOfName IEC_TIMER, OfSystemLibElement IEC_TIMER, OfSystemLibVersion 1.0
"IEC_TIMER"
   // VAR
   //    PT : Time;
   //    ET { ExternalWritable := 'False'} : Time;
   //    IN : Bool;
   //    Q { ExternalWritable := 'False'} : Bool;
   // END_VAR
BEGIN
END_DATA_BLOCK

DATA_BLOCK "TM2"   // DB7
{ S7_Optimized_Access := 'TRUE' }
// stored: AutoNumber true, InstanceOfName IEC_TIMER, OfSystemLibElement IEC_TIMER, OfSystemLibVersion 1.0
"IEC_TIMER"
   // VAR
   //    PT : Time;
   //    ET { ExternalWritable := 'False'} : Time;
   //    IN : Bool;
   //    Q { ExternalWritable := 'False'} : Bool;
   // END_VAR
BEGIN
END_DATA_BLOCK

DATA_BLOCK "TM3"   // DB8
{ S7_Optimized_Access := 'TRUE' }
// stored: AutoNumber true, InstanceOfName IEC_TIMER, OfSystemLibElement IEC_TIMER, OfSystemLibVersion 1.0
"IEC_TIMER"
   // VAR
   //    PT : Time;
   //    ET { ExternalWritable := 'False'} : Time;
   //    IN : Bool;
   //    Q { ExternalWritable := 'False'} : Bool;
   // END_VAR
BEGIN
END_DATA_BLOCK

DATA_BLOCK "TON_Alarme_XV102_1"   // DB16
{ S7_Optimized_Access := 'TRUE' }
// stored: AutoNumber true, InstanceOfName IEC_TIMER, OfSystemLibElement IEC_TIMER, OfSystemLibVersion 1.0
"IEC_TIMER"
   // VAR
   //    PT : Time;
   //    ET { ExternalWritable := 'False'} : Time;
   //    IN : Bool;
   //    Q { ExternalWritable := 'False'} : Bool;
   // END_VAR
BEGIN
END_DATA_BLOCK

DATA_BLOCK "TON_Alarme_XV102_2"   // DB26
{ S7_Optimized_Access := 'TRUE' }
// stored: AutoNumber true, InstanceOfName IEC_TIMER, OfSystemLibElement IEC_TIMER, OfSystemLibVersion 1.0
"IEC_TIMER"
   // VAR
   //    PT : Time;
   //    ET { ExternalWritable := 'False'} : Time;
   //    IN : Bool;
   //    Q { ExternalWritable := 'False'} : Bool;
   // END_VAR
BEGIN
END_DATA_BLOCK

DATA_BLOCK "T_DOS_COAGULANTE"   // DB9
{ S7_Optimized_Access := 'TRUE' }
// stored: AutoNumber true, InstanceOfName IEC_TIMER, OfSystemLibElement IEC_TIMER, OfSystemLibVersion 1.0
"IEC_TIMER"
   // VAR RETAIN
   //    PT : Time;
   //    ET { ExternalWritable := 'False'} : Time;
   //    IN : Bool;
   //    Q { ExternalWritable := 'False'} : Bool;
   // END_VAR
BEGIN
END_DATA_BLOCK

